LIN {X 0,Y 523.988,Z 418.315,A -85,B 0,C 180,E1 -4858.463,E2 -4858.463} C_VEL
LIN {X 0,Y 524.311,Z 419.919,A -85,B 0,C 180,E1 -4858.848,E2 -4858.848} C_VEL
LIN {X 0,Y 524.202,Z 424.484,A -85,B 0,C 180,E1 -4859.928,E2 -4859.928} C_VEL
LIN {X 0,Y 525.991,Z 433.873,A -85,B 0,C 180,E1 -4860.12,E2 -4860.12} C_VEL
LIN {X 0,Y 525.479,Z 529.837,A -85,B 0,C 180,E1 -4861.485,E2 -4861.485} C_VEL
LIN {X 0,Y 525.253,Z 542.81,A -85,B 0,C 180,E1 -4861.821,E2 -4861.821} C_VEL
LIN {X 0,Y 525.093,Z 555.331,A -85,B 0,C 180,E1 -4862.301,E2 -4862.301} C_VEL
LIN {X 0,Y 524.836,Z 568.104,A -85,B 0,C 180,E1 -4862.974,E2 -4862.974} C_VEL
LIN {X 0,Y 524.493,Z 579.334,A -85,B 0,C 180,E1 -4863.745,E2 -4863.745} C_VEL
LIN {X 0,Y 524.25,Z 589.443,A -85,B 0,C 180,E1 -4864.614,E2 -4864.614} C_VEL
LIN {X 0,Y 524.02,Z 598.626,A -85,B 0,C 180,E1 -4865.58,E2 -4865.58} C_VEL
LIN {X 0,Y 523.843,Z 606.368,A -85,B 0,C 180,E1 -4866.58,E2 -4866.58} C_VEL
LIN {X 0,Y 523.721,Z 613.507,A -85,B 0,C 180,E1 -4867.712,E2 -4867.712} C_VEL
LIN {X 0,Y 523.534,Z 619.416,A -85,B 0,C 180,E1 -4868.881,E2 -4868.881} C_VEL
LIN {X 0,Y 523.46,Z 624.093,A -85,B 0,C 180,E1 -4870.052,E2 -4870.052} C_VEL
LIN {X 0,Y 523.411,Z 628.198,A -85,B 0,C 180,E1 -4871.42,E2 -4871.42} C_VEL
LIN {X 0,Y 523.321,Z 630.26,A -85,B 0,C 180,E1 -4872.408,E2 -4872.408} C_VEL
LIN {X 0,Y 523.324,Z 632.229,A -85,B 0,C 180,E1 -4873.989,E2 -4873.989} C_VEL
LIN {X 0,Y 523.299,Z 632.553,A -85,B 0,C 180,E1 -4874.784,E2 -4874.784} C_VEL
LIN {X 0,Y 523.254,Z 631.982,A -85,B 0,C 180,E1 -4876.383,E2 -4876.383} C_VEL
LIN {X 0,Y 523.312,Z 630.501,A -85,B 0,C 180,E1 -4877.536,E2 -4877.536} C_VEL
LIN {X 0,Y 523.374,Z 626.71,A -85,B 0,C 180,E1 -4879.208,E2 -4879.208} C_VEL
LIN {X 0,Y 523.466,Z 622.639,A -85,B 0,C 180,E1 -4880.431,E2 -4880.431} C_VEL
LIN {X 0,Y 523.581,Z 616.177,A -85,B 0,C 180,E1 -4881.869,E2 -4881.869} C_VEL
LIN {X 0,Y 523.697,Z 610.264,A -85,B 0,C 180,E1 -4882.903,E2 -4882.903} C_VEL
LIN {X 0,Y 523.919,Z 602.842,A -85,B 0,C 180,E1 -4883.966,E2 -4883.966} C_VEL
LIN {X 0,Y 524.086,Z 596.098,A -85,B 0,C 180,E1 -4884.775,E2 -4884.775} C_VEL
LIN {X 0,Y 524.315,Z 587.958,A -85,B 0,C 180,E1 -4885.601,E2 -4885.601} C_VEL
LIN {X 0,Y 524.554,Z 577.757,A -85,B 0,C 180,E1 -4886.454,E2 -4886.454} C_VEL
LIN {X 0,Y 524.832,Z 566.75,A -85,B 0,C 180,E1 -4887.192,E2 -4887.192} C_VEL
LIN {X 0,Y 525.129,Z 555.209,A -85,B 0,C 180,E1 -4887.789,E2 -4887.789} C_VEL
LIN {X 0,Y 525.296,Z 542.798,A -85,B 0,C 180,E1 -4888.267,E2 -4888.267} C_VEL
LIN {X 0,Y 525.449,Z 530.555,A -85,B 0,C 180,E1 -4888.593,E2 -4888.593} C_VEL
LIN {X 0,Y 525.677,Z 483.88,A -85,B 0,C 180,E1 -4889.263,E2 -4889.263} C_VEL
LIN {X 0,Y 525.84,Z 432.621,A -85,B 0,C 180,E1 -4889.982,E2 -4889.982} C_VEL
LIN {X 0,Y 525.253,Z 429.53,A -85,B 0,C 180,E1 -4890.045,E2 -4890.045} C_VEL
LIN {X 0,Y 524.217,Z 426.571,A -85,B 0,C 180,E1 -4890.171,E2 -4890.171} C_VEL
LIN {X 0,Y 521.978,Z 423.441,A -85,B 0,C 180,E1 -4890.485,E2 -4890.485} C_VEL
LIN {X 0,Y 519.924,Z 421.666,A -85,B 0,C 180,E1 -4890.834,E2 -4890.834} C_VEL
LIN {X 0,Y 517.617,Z 419.8,A -85,B 0,C 180,E1 -4891.394,E2 -4891.394} C_VEL
LIN {X 0,Y 516.936,Z 419.124,A -85,B 0,C 180,E1 -4891.783,E2 -4891.783} C_VEL
LIN {X 0,Y 516.908,Z 419.099,A -85,B 0,C 180,E1 -4891.864,E2 -4891.864} C_VEL
LIN {X 0,Y 516.875,Z 419.099,A -85,B 0,C 180,E1 -4894.825,E2 -4894.825} C_VEL
LIN {X 0,Y 516.867,Z 419.099,A -85,B 0,C 180,E1 -4897.94,E2 -4897.94} C_VEL
LIN {X 0,Y 516.856,Z 419.102,A -85,B 0,C 180,E1 -4900.744,E2 -4900.744} C_VEL
LIN {X 0,Y 516.884,Z 419.097,A -85,B 0,C 180,E1 -4903.903,E2 -4903.903} C_VEL
LIN {X 0,Y 516.882,Z 419.099,A -85,B 0,C 180,E1 -4906.107,E2 -4906.107} C_VEL
LIN {X 0,Y 516.854,Z 419.098,A -85,B 0,C 180,E1 -4909.255,E2 -4909.255} C_VEL
LIN {X 0,Y 516.864,Z 419.101,A -85,B 0,C 180,E1 -4912.06,E2 -4912.06} C_VEL
LIN {X 0,Y 516.876,Z 419.096,A -85,B 0,C 180,E1 -4915.174,E2 -4915.174} C_VEL
LIN {X 0,Y 516.875,Z 419.098,A -85,B 0,C 180,E1 -4917.975,E2 -4917.975} C_VEL
LIN {X 0,Y 516.906,Z 419.097,A -85,B 0,C 180,E1 -4920.694,E2 -4920.694} C_VEL
LIN {X 0,Y 516.89,Z 419.095,A -85,B 0,C 180,E1 -4923.816,E2 -4923.816} C_VEL
LIN {X 0,Y 516.86,Z 419.102,A -85,B 0,C 180,E1 -4926.776,E2 -4926.776} C_VEL
LIN {X 0,Y 516.94,Z 419.088,A -85,B 0,C 180,E1 -4929.732,E2 -4929.732} C_VEL
LIN {X 0,Y 516.887,Z 419.101,A -85,B 0,C 180,E1 -4932.594,E2 -4932.594} C_VEL
LIN {X 0,Y 516.938,Z 419.089,A -85,B 0,C 180,E1 -4935.03,E2 -4935.03} C_VEL
LIN {X 0,Y 516.969,Z 419.089,A -85,B 0,C 180,E1 -4938.233,E2 -4938.233} C_VEL
LIN {X 0,Y 516.955,Z 419.085,A -85,B 0,C 180,E1 -4941.399,E2 -4941.399} C_VEL
LIN {X 0,Y 517.014,Z 419.087,A -85,B 0,C 180,E1 -4944.54,E2 -4944.54} C_VEL
LIN {X 0,Y 517.082,Z 419.07,A -85,B 0,C 180,E1 -4947.663,E2 -4947.663} C_VEL
LIN {X 0,Y 517.092,Z 419.073,A -85,B 0,C 180,E1 -4950.778,E2 -4950.778} C_VEL
LIN {X 0,Y 516.974,Z 419.084,A -85,B 0,C 180,E1 -4953.117,E2 -4953.117} C_VEL
LIN {X 0,Y 517.008,Z 419.084,A -85,B 0,C 180,E1 -4956.243,E2 -4956.243} C_VEL
LIN {X 0,Y 516.94,Z 419.087,A -85,B 0,C 180,E1 -4959.389,E2 -4959.389} C_VEL
LIN {X 0,Y 516.954,Z 419.086,A -85,B 0,C 180,E1 -4961.807,E2 -4961.807} C_VEL
LIN {X 0,Y 516.949,Z 419.087,A -85,B 0,C 180,E1 -4965.147,E2 -4965.147} C_VEL
LIN {X 0,Y 516.917,Z 419.095,A -85,B 0,C 180,E1 -4968.222,E2 -4968.222} C_VEL
LIN {X 0,Y 516.913,Z 419.097,A -85,B 0,C 180,E1 -4970.701,E2 -4970.701} C_VEL
LIN {X 0,Y 516.891,Z 419.096,A -85,B 0,C 180,E1 -4974.073,E2 -4974.073} C_VEL
LIN {X 0,Y 516.897,Z 419.1,A -85,B 0,C 180,E1 -4976.659,E2 -4976.659} C_VEL
LIN {X 0,Y 516.91,Z 419.091,A -85,B 0,C 180,E1 -4979.523,E2 -4979.523} C_VEL
LIN {X 0,Y 516.896,Z 419.102,A -85,B 0,C 180,E1 -4982.543,E2 -4982.543} C_VEL
LIN {X 0,Y 516.864,Z 419.097,A -85,B 0,C 180,E1 -4985.329,E2 -4985.329} C_VEL
LIN {X 0,Y 516.878,Z 419.096,A -85,B 0,C 180,E1 -4987.943,E2 -4987.943} C_VEL
LIN {X 0,Y 516.881,Z 419.101,A -85,B 0,C 180,E1 -4990.742,E2 -4990.742} C_VEL
LIN {X 0,Y 516.88,Z 419.096,A -85,B 0,C 180,E1 -4993.903,E2 -4993.903} C_VEL
LIN {X 0,Y 516.88,Z 419.097,A -85,B 0,C 180,E1 -4996.107,E2 -4996.107} C_VEL
LIN {X 0,Y 516.881,Z 419.095,A -85,B 0,C 180,E1 -4999.258,E2 -4999.258} C_VEL
LIN {X 0,Y 516.86,Z 419.102,A -85,B 0,C 180,E1 -5002.274,E2 -5002.274} C_VEL
LIN {X 0,Y 516.881,Z 419.096,A -85,B 0,C 180,E1 -5005.175,E2 -5005.175} C_VEL
LIN {X 0,Y 516.873,Z 419.097,A -85,B 0,C 180,E1 -5007.975,E2 -5007.975} C_VEL
LIN {X 0,Y 516.92,Z 419.098,A -85,B 0,C 180,E1 -5010.695,E2 -5010.695} C_VEL
LIN {X 0,Y 516.911,Z 419.091,A -85,B 0,C 180,E1 -5013.811,E2 -5013.811} C_VEL
LIN {X 0,Y 516.86,Z 419.104,A -85,B 0,C 180,E1 -5016.776,E2 -5016.776} C_VEL
LIN {X 0,Y 516.939,Z 419.087,A -85,B 0,C 180,E1 -5019.732,E2 -5019.732} C_VEL
LIN {X 0,Y 516.905,Z 419.101,A -85,B 0,C 180,E1 -5022.595,E2 -5022.595} C_VEL
LIN {X 0,Y 516.941,Z 419.09,A -85,B 0,C 180,E1 -5025.03,E2 -5025.03} C_VEL
LIN {X 0,Y 516.966,Z 419.087,A -85,B 0,C 180,E1 -5028.234,E2 -5028.234} C_VEL
LIN {X 0,Y 516.965,Z 419.085,A -85,B 0,C 180,E1 -5031.4,E2 -5031.4} C_VEL
LIN {X 0,Y 517.025,Z 419.085,A -85,B 0,C 180,E1 -5034.54,E2 -5034.54} C_VEL
LIN {X 0,Y 517.083,Z 419.069,A -85,B 0,C 180,E1 -5037.663,E2 -5037.663} C_VEL
LIN {X 0,Y 517.093,Z 419.076,A -85,B 0,C 180,E1 -5040.779,E2 -5040.779} C_VEL
LIN {X 0,Y 517.009,Z 419.081,A -85,B 0,C 180,E1 -5043.117,E2 -5043.117} C_VEL
LIN {X 0,Y 517.008,Z 419.082,A -85,B 0,C 180,E1 -5046.243,E2 -5046.243} C_VEL
LIN {X 0,Y 516.944,Z 419.087,A -85,B 0,C 180,E1 -5049.389,E2 -5049.389} C_VEL
LIN {X 0,Y 516.952,Z 419.086,A -85,B 0,C 180,E1 -5051.807,E2 -5051.807} C_VEL
LIN {X 0,Y 516.948,Z 419.089,A -85,B 0,C 180,E1 -5055.148,E2 -5055.148} C_VEL
LIN {X 0,Y 516.916,Z 419.093,A -85,B 0,C 180,E1 -5058.223,E2 -5058.223} C_VEL
LIN {X 0,Y 516.912,Z 419.1,A -85,B 0,C 180,E1 -5060.702,E2 -5060.702} C_VEL
LIN {X 0,Y 516.902,Z 419.093,A -85,B 0,C 180,E1 -5064.073,E2 -5064.073} C_VEL
LIN {X 0,Y 516.904,Z 419.101,A -85,B 0,C 180,E1 -5066.659,E2 -5066.659} C_VEL
LIN {X 0,Y 516.911,Z 419.091,A -85,B 0,C 180,E1 -5069.524,E2 -5069.524} C_VEL
LIN {X 0,Y 516.895,Z 419.099,A -85,B 0,C 180,E1 -5072.543,E2 -5072.543} C_VEL
LIN {X 0,Y 516.867,Z 419.098,A -85,B 0,C 180,E1 -5075.33,E2 -5075.33} C_VEL
LIN {X 0,Y 516.88,Z 419.095,A -85,B 0,C 180,E1 -5077.943,E2 -5077.943} C_VEL
LIN {X 0,Y 516.883,Z 419.104,A -85,B 0,C 180,E1 -5080.742,E2 -5080.742} C_VEL
LIN {X 0,Y 516.883,Z 419.102,A -85,B 0,C 180,E1 -5082.832,E2 -5082.832} C_VEL
LIN {X 0,Y 516.924,Z 419.094,A -85,B 0,C 180,E1 -5085.01,E2 -5085.01} C_VEL
LIN {X 0,Y 516.914,Z 419.095,A -85,B 0,C 180,E1 -5088.399,E2 -5088.399} C_VEL
LIN {X 0,Y 516.882,Z 419.096,A -85,B 0,C 180,E1 -5091.284,E2 -5091.284} C_VEL
LIN {X 0,Y 516.869,Z 419.098,A -85,B 0,C 180,E1 -5094.22,E2 -5094.22} C_VEL
LIN {X 0,Y 516.896,Z 419.098,A -85,B 0,C 180,E1 -5097.053,E2 -5097.053} C_VEL
LIN {X 0,Y 516.893,Z 419.094,A -85,B 0,C 180,E1 -5099.797,E2 -5099.797} C_VEL
LIN {X 0,Y 516.925,Z 419.097,A -85,B 0,C 180,E1 -5102.467,E2 -5102.467} C_VEL
LIN {X 0,Y 516.954,Z 419.122,A -85,B 0,C 180,E1 -5103.438,E2 -5103.438} C_VEL
LIN {X 0,Y 519.032,Z 430.297,A -85,B 0,C 180,E1 -5105.181,E2 -5105.181} C_VEL
LIN {X 0,Y 518.58,Z 445.899,A -85,B 0,C 180,E1 -5107.421,E2 -5107.421} C_VEL
LIN {X 0,Y 518.088,Z 466.974,A -85,B 0,C 180,E1 -5110.383,E2 -5110.383} C_VEL
LIN {X 0,Y 517.598,Z 488.869,A -85,B 0,C 180,E1 -5113.433,E2 -5113.433} C_VEL
LIN {X 0,Y 517.403,Z 497.471,A -85,B 0,C 180,E1 -5114.627,E2 -5114.627} C_VEL
LIN {X 0,Y 518.961,Z 510.132,A -85,B 0,C 180,E1 -5114.873,E2 -5114.873} C_VEL
LIN {X 0,Y 518.553,Z 604.493,A -85,B 0,C 180,E1 -5116.205,E2 -5116.205} C_VEL
LIN {X 0,Y 518.352,Z 617.14,A -85,B 0,C 180,E1 -5116.5,E2 -5116.5} C_VEL
LIN {X 0,Y 518.062,Z 630.067,A -85,B 0,C 180,E1 -5116.966,E2 -5116.966} C_VEL
LIN {X 0,Y 517.822,Z 642.684,A -85,B 0,C 180,E1 -5117.594,E2 -5117.594} C_VEL
LIN {X 0,Y 517.526,Z 654.284,A -85,B 0,C 180,E1 -5118.346,E2 -5118.346} C_VEL
LIN {X 0,Y 517.212,Z 665.109,A -85,B 0,C 180,E1 -5119.232,E2 -5119.232} C_VEL
LIN {X 0,Y 516.948,Z 674.862,A -85,B 0,C 180,E1 -5120.216,E2 -5120.216} C_VEL
LIN {X 0,Y 516.739,Z 682.861,A -85,B 0,C 180,E1 -5121.199,E2 -5121.199} C_VEL
LIN {X 0,Y 516.555,Z 690.676,A -85,B 0,C 180,E1 -5122.377,E2 -5122.377} C_VEL
LIN {X 0,Y 516.421,Z 696.438,A -85,B 0,C 180,E1 -5123.446,E2 -5123.446} C_VEL
LIN {X 0,Y 516.402,Z 701.206,A -85,B 0,C 180,E1 -5124.534,E2 -5124.534} C_VEL
LIN {X 0,Y 516.331,Z 705.226,A -85,B 0,C 180,E1 -5125.707,E2 -5125.707} C_VEL
LIN {X 0,Y 516.282,Z 708.192,A -85,B 0,C 180,E1 -5126.879,E2 -5126.879} C_VEL
LIN {X 0,Y 516.261,Z 709.605,A -85,B 0,C 180,E1 -5127.66,E2 -5127.66} C_VEL
LIN {X 0,Y 516.169,Z 711.22,A -85,B 0,C 180,E1 -5129.22,E2 -5129.22} C_VEL
LIN {X 0,Y 516.167,Z 711.435,A -85,B 0,C 180,E1 -5130,E2 -5130} C_VEL
LIN {X 0,Y 516.17,Z 711.214,A -85,B 0,C 180,E1 -5130.78,E2 -5130.78} C_VEL
LIN {X 0,Y 516.261,Z 709.591,A -85,B 0,C 180,E1 -5132.341,E2 -5132.341} C_VEL
LIN {X 0,Y 516.296,Z 708.169,A -85,B 0,C 180,E1 -5133.122,E2 -5133.122} C_VEL
LIN {X 0,Y 516.348,Z 705.187,A -85,B 0,C 180,E1 -5134.293,E2 -5134.293} C_VEL
LIN {X 0,Y 516.402,Z 701.146,A -85,B 0,C 180,E1 -5135.467,E2 -5135.467} C_VEL
LIN {X 0,Y 516.484,Z 695.108,A -85,B 0,C 180,E1 -5136.803,E2 -5136.803} C_VEL
LIN {X 0,Y 516.606,Z 688.128,A -85,B 0,C 180,E1 -5138.016,E2 -5138.016} C_VEL
LIN {X 0,Y 516.8,Z 679.686,A -85,B 0,C 180,E1 -5139.195,E2 -5139.195} C_VEL
LIN {X 0,Y 517.041,Z 671.016,A -85,B 0,C 180,E1 -5140.178,E2 -5140.178} C_VEL
LIN {X 0,Y 517.331,Z 660.315,A -85,B 0,C 180,E1 -5141.163,E2 -5141.163} C_VEL
LIN {X 0,Y 517.576,Z 649.28,A -85,B 0,C 180,E1 -5141.98,E2 -5141.98} C_VEL
LIN {X 0,Y 517.929,Z 637.022,A -85,B 0,C 180,E1 -5142.689,E2 -5142.689} C_VEL
LIN {X 0,Y 518.168,Z 624.585,A -85,B 0,C 180,E1 -5143.231,E2 -5143.231} C_VEL
LIN {X 0,Y 518.419,Z 611.883,A -85,B 0,C 180,E1 -5143.624,E2 -5143.624} C_VEL
LIN {X 0,Y 518.649,Z 597.089,A -85,B 0,C 180,E1 -5143.893,E2 -5143.893} C_VEL
LIN {X 0,Y 518.808,Z 507.894,A -85,B 0,C 180,E1 -5145.156,E2 -5145.156} C_VEL
LIN {X 0,Y 517.345,Z 496.789,A -85,B 0,C 180,E1 -5145.376,E2 -5145.376} C_VEL
LIN {X 0,Y 517.74,Z 476.234,A -85,B 0,C 180,E1 -5148.193,E2 -5148.193} C_VEL
LIN {X 0,Y 518.264,Z 454.035,A -85,B 0,C 180,E1 -5151.269,E2 -5151.269} C_VEL
LIN {X 0,Y 518.756,Z 431.819,A -85,B 0,C 180,E1 -5154.407,E2 -5154.407} C_VEL
LIN {X 0,Y 518.806,Z 428.851,A -85,B 0,C 180,E1 -5154.831,E2 -5154.831} C_VEL
LIN {X 0,Y 516.94,Z 419.094,A -85,B 0,C 180,E1 -5156.352,E2 -5156.352} C_VEL
LIN {X 0,Y 516.915,Z 419.098,A -85,B 0,C 180,E1 -5159.524,E2 -5159.524} C_VEL
LIN {X 0,Y 516.9,Z 419.1,A -85,B 0,C 180,E1 -5162.544,E2 -5162.544} C_VEL
LIN {X 0,Y 516.872,Z 419.103,A -85,B 0,C 180,E1 -5165.33,E2 -5165.33} C_VEL
LIN {X 0,Y 516.884,Z 419.096,A -85,B 0,C 180,E1 -5167.943,E2 -5167.943} C_VEL
LIN {X 0,Y 516.887,Z 419.102,A -85,B 0,C 180,E1 -5170.742,E2 -5170.742} C_VEL
LIN {X 0,Y 516.886,Z 419.104,A -85,B 0,C 180,E1 -5172.832,E2 -5172.832} C_VEL
LIN {X 0,Y 516.899,Z 419.098,A -85,B 0,C 180,E1 -5175.007,E2 -5175.007} C_VEL
LIN {X 0,Y 516.914,Z 419.097,A -85,B 0,C 180,E1 -5178.399,E2 -5178.399} C_VEL
LIN {X 0,Y 516.883,Z 419.096,A -85,B 0,C 180,E1 -5181.284,E2 -5181.284} C_VEL
LIN {X 0,Y 516.87,Z 419.101,A -85,B 0,C 180,E1 -5184.219,E2 -5184.219} C_VEL
LIN {X 0,Y 516.899,Z 419.094,A -85,B 0,C 180,E1 -5187.053,E2 -5187.053} C_VEL
LIN {X 0,Y 516.871,Z 419.098,A -85,B 0,C 180,E1 -5189.795,E2 -5189.795} C_VEL
LIN {X 0,Y 516.877,Z 419.104,A -85,B 0,C 180,E1 -5192.464,E2 -5192.464} C_VEL
LIN {X 0,Y 516.848,Z 419.101,A -85,B 0,C 180,E1 -5195.069,E2 -5195.069} C_VEL
LIN {X 0,Y 516.873,Z 419.099,A -85,B 0,C 180,E1 -5197.622,E2 -5197.622} C_VEL
LIN {X 0,Y 516.866,Z 419.105,A -85,B 0,C 180,E1 -5200.127,E2 -5200.127} C_VEL
LIN {X 0,Y 516.867,Z 419.1,A -85,B 0,C 180,E1 -5202.594,E2 -5202.594} C_VEL
LIN {X 0,Y 516.857,Z 419.106,A -85,B 0,C 180,E1 -5205.832,E2 -5205.832} C_VEL
LIN {X 0,Y 516.923,Z 419.097,A -85,B 0,C 180,E1 -5208.233,E2 -5208.233} C_VEL
LIN {X 0,Y 516.92,Z 419.095,A -85,B 0,C 180,E1 -5211.399,E2 -5211.399} C_VEL
LIN {X 0,Y 516.98,Z 419.087,A -85,B 0,C 180,E1 -5214.539,E2 -5214.539} C_VEL
LIN {X 0,Y 517.025,Z 419.086,A -85,B 0,C 180,E1 -5218.052,E2 -5218.052} C_VEL
LIN {X 0,Y 517.007,Z 419.337,A -85,B 0,C 180,E1 -5218.345,E2 -5218.345} C_VEL
LIN {X 0,Y 517.28,Z 423.009,A -85,B 0,C 180,E1 -5219.221,E2 -5219.221} C_VEL
LIN {X 0,Y 517.308,Z 425.389,A -85,B 0,C 180,E1 -5219.732,E2 -5219.732} C_VEL
LIN {X 0,Y 519.149,Z 434.62,A -85,B 0,C 180,E1 -5219.927,E2 -5219.927} C_VEL
LIN {X 0,Y 518.51,Z 531.284,A -85,B 0,C 180,E1 -5221.335,E2 -5221.335} C_VEL
LIN {X 0,Y 518.342,Z 544.694,A -85,B 0,C 180,E1 -5221.7,E2 -5221.7} C_VEL
LIN {X 0,Y 518.14,Z 556.874,A -85,B 0,C 180,E1 -5222.186,E2 -5222.186} C_VEL
LIN {X 0,Y 517.904,Z 568.571,A -85,B 0,C 180,E1 -5222.82,E2 -5222.82} C_VEL
LIN {X 0,Y 517.551,Z 579.85,A -85,B 0,C 180,E1 -5223.601,E2 -5223.601} C_VEL
LIN {X 0,Y 517.273,Z 589.985,A -85,B 0,C 180,E1 -5224.481,E2 -5224.481} C_VEL
LIN {X 0,Y 517.038,Z 599.151,A -85,B 0,C 180,E1 -5225.46,E2 -5225.46} C_VEL
LIN {X 0,Y 516.797,Z 607.986,A -85,B 0,C 180,E1 -5226.632,E2 -5226.632} C_VEL
LIN {X 0,Y 516.641,Z 615.138,A -85,B 0,C 180,E1 -5227.818,E2 -5227.818} C_VEL
LIN {X 0,Y 516.488,Z 620.854,A -85,B 0,C 180,E1 -5229.003,E2 -5229.003} C_VEL
LIN {X 0,Y 516.4,Z 625.362,A -85,B 0,C 180,E1 -5230.191,E2 -5230.191} C_VEL
LIN {X 0,Y 516.302,Z 629.7,A -85,B 0,C 180,E1 -5231.782,E2 -5231.782} C_VEL
LIN {X 0,Y 516.24,Z 631.194,A -85,B 0,C 180,E1 -5232.581,E2 -5232.581} C_VEL
LIN {X 0,Y 516.244,Z 632.889,A -85,B 0,C 180,E1 -5234.185,E2 -5234.185} C_VEL
LIN {X 0,Y 516.21,Z 633.139,A -85,B 0,C 180,E1 -5234.992,E2 -5234.992} C_VEL
LIN {X 0,Y 516.195,Z 632.919,A -85,B 0,C 180,E1 -5235.801,E2 -5235.801} C_VEL
LIN {X 0,Y 516.241,Z 631.278,A -85,B 0,C 180,E1 -5237.428,E2 -5237.428} C_VEL
LIN {X 0,Y 516.296,Z 628.843,A -85,B 0,C 180,E1 -5238.656,E2 -5238.656} C_VEL
LIN {X 0,Y 516.357,Z 625.294,A -85,B 0,C 180,E1 -5239.893,E2 -5239.893} C_VEL
LIN {X 0,Y 516.445,Z 620.518,A -85,B 0,C 180,E1 -5241.138,E2 -5241.138} C_VEL
LIN {X 0,Y 516.605,Z 614.367,A -85,B 0,C 180,E1 -5242.391,E2 -5242.391} C_VEL
LIN {X 0,Y 516.818,Z 606.511,A -85,B 0,C 180,E1 -5243.651,E2 -5243.651} C_VEL
LIN {X 0,Y 517.042,Z 597.84,A -85,B 0,C 180,E1 -5244.76,E2 -5244.76} C_VEL
LIN {X 0,Y 517.309,Z 589.228,A -85,B 0,C 180,E1 -5245.661,E2 -5245.661} C_VEL
LIN {X 0,Y 517.54,Z 579.353,A -85,B 0,C 180,E1 -5246.513,E2 -5246.513} C_VEL
LIN {X 0,Y 517.846,Z 568.558,A -85,B 0,C 180,E1 -5247.261,E2 -5247.261} C_VEL
LIN {X 0,Y 518.187,Z 556.468,A -85,B 0,C 180,E1 -5247.915,E2 -5247.915} C_VEL
LIN {X 0,Y 518.404,Z 544.005,A -85,B 0,C 180,E1 -5248.409,E2 -5248.409} C_VEL
LIN {X 0,Y 518.543,Z 531.159,A -85,B 0,C 180,E1 -5248.76,E2 -5248.76} C_VEL
LIN {X 0,Y 518.771,Z 491.313,A -85,B 0,C 180,E1 -5249.348,E2 -5249.348} C_VEL
LIN {X 0,Y 518.956,Z 433.244,A -85,B 0,C 180,E1 -5250.182,E2 -5250.182} C_VEL
LIN {X 0,Y 517.154,Z 424.213,A -85,B 0,C 180,E1 -5250.384,E2 -5250.384} C_VEL
LIN {X 0,Y 516.963,Z 419.316,A -85,B 0,C 180,E1 -5251.497,E2 -5251.497} C_VEL
LIN {X 0,Y 516.908,Z 419.099,A -85,B 0,C 180,E1 -5251.864,E2 -5251.864} C_VEL
LIN {X 0,Y 516.206,Z 419.188,A -85,B 0,C 180,E1 -5252.514,E2 -5252.514} C_VEL
LIN {X 0,Y 513.315,Z 419.546,A -85,B 0,C 180,E1 -5253.57,E2 -5253.57} C_VEL
LIN {X 0,Y 510.903,Z 419.848,A -85,B 0,C 180,E1 -5254.42,E2 -5254.42} C_VEL
LIN {X 0,Y 509.889,Z 419.968,A -85,B 0,C 180,E1 -5255.077,E2 -5255.077} C_VEL
LIN {X 0,Y 509.816,Z 419.976,A -85,B 0,C 180,E1 -5255.299,E2 -5255.299} C_VEL
LIN {X 0,Y 509.819,Z 419.983,A -85,B 0,C 180,E1 -5258.341,E2 -5258.341} C_VEL
LIN {X 0,Y 509.834,Z 419.972,A -85,B 0,C 180,E1 -5261.428,E2 -5261.428} C_VEL
LIN {X 0,Y 509.842,Z 419.977,A -85,B 0,C 180,E1 -5264.67,E2 -5264.67} C_VEL
LIN {X 0,Y 509.793,Z 419.978,A -85,B 0,C 180,E1 -5267.505,E2 -5267.505} C_VEL
LIN {X 0,Y 509.834,Z 419.978,A -85,B 0,C 180,E1 -5270.646,E2 -5270.646} C_VEL
LIN {X 0,Y 509.783,Z 419.979,A -85,B 0,C 180,E1 -5273.643,E2 -5273.643} C_VEL
LIN {X 0,Y 509.854,Z 419.978,A -85,B 0,C 180,E1 -5276.538,E2 -5276.538} C_VEL
LIN {X 0,Y 509.836,Z 419.972,A -85,B 0,C 180,E1 -5279.333,E2 -5279.333} C_VEL
LIN {X 0,Y 509.838,Z 419.976,A -85,B 0,C 180,E1 -5282.051,E2 -5282.051} C_VEL
LIN {X 0,Y 509.808,Z 419.981,A -85,B 0,C 180,E1 -5284.7,E2 -5284.7} C_VEL
LIN {X 0,Y 509.828,Z 419.973,A -85,B 0,C 180,E1 -5287.458,E2 -5287.458} C_VEL
LIN {X 0,Y 509.917,Z 419.964,A -85,B 0,C 180,E1 -5289.844,E2 -5289.844} C_VEL
LIN {X 0,Y 509.849,Z 419.971,A -85,B 0,C 180,E1 -5293.173,E2 -5293.173} C_VEL
LIN {X 0,Y 509.854,Z 419.97,A -85,B 0,C 180,E1 -5295.634,E2 -5295.634} C_VEL
LIN {X 0,Y 509.914,Z 419.966,A -85,B 0,C 180,E1 -5298.874,E2 -5298.874} C_VEL
LIN {X 0,Y 509.91,Z 419.966,A -85,B 0,C 180,E1 -5302.077,E2 -5302.077} C_VEL
LIN {X 0,Y 509.965,Z 419.966,A -85,B 0,C 180,E1 -5304.464,E2 -5304.464} C_VEL
LIN {X 0,Y 510.051,Z 419.945,A -85,B 0,C 180,E1 -5307.631,E2 -5307.631} C_VEL
LIN {X 0,Y 510.062,Z 419.949,A -85,B 0,C 180,E1 -5310.789,E2 -5310.789} C_VEL
LIN {X 0,Y 509.918,Z 419.963,A -85,B 0,C 180,E1 -5313.16,E2 -5313.16} C_VEL
LIN {X 0,Y 509.977,Z 419.961,A -85,B 0,C 180,E1 -5316.329,E2 -5316.329} C_VEL
LIN {X 0,Y 509.88,Z 419.967,A -85,B 0,C 180,E1 -5319.52,E2 -5319.52} C_VEL
LIN {X 0,Y 509.906,Z 419.965,A -85,B 0,C 180,E1 -5321.931,E2 -5321.931} C_VEL
LIN {X 0,Y 509.896,Z 419.965,A -85,B 0,C 180,E1 -5325.241,E2 -5325.241} C_VEL
LIN {X 0,Y 509.862,Z 419.978,A -85,B 0,C 180,E1 -5328.483,E2 -5328.483} C_VEL
LIN {X 0,Y 509.851,Z 419.973,A -85,B 0,C 180,E1 -5331.001,E2 -5331.001} C_VEL
LIN {X 0,Y 509.823,Z 419.974,A -85,B 0,C 180,E1 -5333.564,E2 -5333.564} C_VEL
LIN {X 0,Y 509.879,Z 419.974,A -85,B 0,C 180,E1 -5336.371,E2 -5336.371} C_VEL
LIN {X 0,Y 509.859,Z 419.97,A -85,B 0,C 180,E1 -5339.726,E2 -5339.726} C_VEL
LIN {X 0,Y 509.873,Z 419.973,A -85,B 0,C 180,E1 -5342.774,E2 -5342.774} C_VEL
LIN {X 0,Y 509.823,Z 419.974,A -85,B 0,C 180,E1 -5345.578,E2 -5345.578} C_VEL
LIN {X 0,Y 509.848,Z 419.977,A -85,B 0,C 180,E1 -5348.338,E2 -5348.338} C_VEL
LIN {X 0,Y 509.852,Z 419.97,A -85,B 0,C 180,E1 -5351.426,E2 -5351.426} C_VEL
LIN {X 0,Y 509.838,Z 419.98,A -85,B 0,C 180,E1 -5354.67,E2 -5354.67} C_VEL
LIN {X 0,Y 509.849,Z 419.973,A -85,B 0,C 180,E1 -5358.104,E2 -5358.104} C_VEL
LIN {X 0,Y 509.845,Z 419.979,A -85,B 0,C 180,E1 -5360.647,E2 -5360.647} C_VEL
LIN {X 0,Y 509.808,Z 419.976,A -85,B 0,C 180,E1 -5363.645,E2 -5363.645} C_VEL
LIN {X 0,Y 509.858,Z 419.978,A -85,B 0,C 180,E1 -5366.539,E2 -5366.539} C_VEL
LIN {X 0,Y 509.845,Z 419.972,A -85,B 0,C 180,E1 -5369.334,E2 -5369.334} C_VEL
LIN {X 0,Y 509.882,Z 419.968,A -85,B 0,C 180,E1 -5372.054,E2 -5372.054} C_VEL
LIN {X 0,Y 509.824,Z 419.982,A -85,B 0,C 180,E1 -5374.701,E2 -5374.701} C_VEL
LIN {X 0,Y 509.826,Z 419.974,A -85,B 0,C 180,E1 -5377.458,E2 -5377.458} C_VEL
LIN {X 0,Y 509.916,Z 419.963,A -85,B 0,C 180,E1 -5379.845,E2 -5379.845} C_VEL
LIN {X 0,Y 509.87,Z 419.97,A -85,B 0,C 180,E1 -5383.174,E2 -5383.174} C_VEL
LIN {X 0,Y 509.861,Z 419.969,A -85,B 0,C 180,E1 -5385.634,E2 -5385.634} C_VEL
LIN {X 0,Y 509.912,Z 419.968,A -85,B 0,C 180,E1 -5388.875,E2 -5388.875} C_VEL
LIN {X 0,Y 509.951,Z 419.96,A -85,B 0,C 180,E1 -5392.078,E2 -5392.078} C_VEL
LIN {X 0,Y 509.976,Z 419.961,A -85,B 0,C 180,E1 -5394.464,E2 -5394.464} C_VEL
LIN {X 0,Y 510.054,Z 419.945,A -85,B 0,C 180,E1 -5397.631,E2 -5397.631} C_VEL
LIN {X 0,Y 510.063,Z 419.951,A -85,B 0,C 180,E1 -5400.79,E2 -5400.79} C_VEL
LIN {X 0,Y 509.95,Z 419.96,A -85,B 0,C 180,E1 -5403.16,E2 -5403.16} C_VEL
LIN {X 0,Y 509.977,Z 419.959,A -85,B 0,C 180,E1 -5406.33,E2 -5406.33} C_VEL
LIN {X 0,Y 509.911,Z 419.972,A -85,B 0,C 180,E1 -5408.72,E2 -5408.72} C_VEL
LIN {X 0,Y 509.905,Z 419.964,A -85,B 0,C 180,E1 -5411.932,E2 -5411.932} C_VEL
LIN {X 0,Y 509.894,Z 419.967,A -85,B 0,C 180,E1 -5415.242,E2 -5415.242} C_VEL
LIN {X 0,Y 509.867,Z 419.969,A -85,B 0,C 180,E1 -5417.993,E2 -5417.993} C_VEL
LIN {X 0,Y 509.887,Z 419.971,A -85,B 0,C 180,E1 -5420.402,E2 -5420.402} C_VEL
LIN {X 0,Y 509.829,Z 419.973,A -85,B 0,C 180,E1 -5423.564,E2 -5423.564} C_VEL
LIN {X 0,Y 509.886,Z 419.97,A -85,B 0,C 180,E1 -5426.373,E2 -5426.373} C_VEL
LIN {X 0,Y 509.872,Z 419.975,A -85,B 0,C 180,E1 -5428.845,E2 -5428.845} C_VEL
LIN {X 0,Y 509.82,Z 419.974,A -85,B 0,C 180,E1 -5431.59,E2 -5431.59} C_VEL
LIN {X 0,Y 509.848,Z 419.975,A -85,B 0,C 180,E1 -5434.414,E2 -5434.414} C_VEL
LIN {X 0,Y 509.817,Z 419.976,A -85,B 0,C 180,E1 -5437.341,E2 -5437.341} C_VEL
LIN {X 0,Y 509.838,Z 419.976,A -85,B 0,C 180,E1 -5440.382,E2 -5440.382} C_VEL
LIN {X 0,Y 509.823,Z 419.978,A -85,B 0,C 180,E1 -5443.062,E2 -5443.062} C_VEL
LIN {X 0,Y 509.831,Z 419.973,A -85,B 0,C 180,E1 -5445.793,E2 -5445.793} C_VEL
LIN {X 0,Y 509.856,Z 419.976,A -85,B 0,C 180,E1 -5448.575,E2 -5448.575} C_VEL
LIN {X 0,Y 509.851,Z 419.97,A -85,B 0,C 180,E1 -5451.787,E2 -5451.787} C_VEL
LIN {X 0,Y 509.828,Z 419.98,A -85,B 0,C 180,E1 -5454.622,E2 -5454.622} C_VEL
LIN {X 0,Y 509.862,Z 419.97,A -85,B 0,C 180,E1 -5457.481,E2 -5457.481} C_VEL
LIN {X 0,Y 509.86,Z 419.973,A -85,B 0,C 180,E1 -5460.274,E2 -5460.274} C_VEL
LIN {X 0,Y 509.939,Z 420.148,A -85,B 0,C 180,E1 -5463.258,E2 -5463.258} C_VEL
LIN {X 0,Y 512.148,Z 431.593,A -85,B 0,C 180,E1 -5465.071,E2 -5465.071} C_VEL
LIN {X 0,Y 511.609,Z 447.435,A -85,B 0,C 180,E1 -5467.379,E2 -5467.379} C_VEL
LIN {X 0,Y 511.109,Z 468.029,A -85,B 0,C 180,E1 -5470.313,E2 -5470.313} C_VEL
LIN {X 0,Y 510.548,Z 489.844,A -85,B 0,C 180,E1 -5473.403,E2 -5473.403} C_VEL
LIN {X 0,Y 510.369,Z 496.977,A -85,B 0,C 180,E1 -5474.407,E2 -5474.407} C_VEL
LIN {X 0,Y 512.09,Z 510.248,A -85,B 0,C 180,E1 -5474.674,E2 -5474.674} C_VEL
LIN {X 0,Y 511.66,Z 603.258,A -85,B 0,C 180,E1 -5476.016,E2 -5476.016} C_VEL
LIN {X 0,Y 511.438,Z 616.185,A -85,B 0,C 180,E1 -5476.313,E2 -5476.313} C_VEL
LIN {X 0,Y 511.134,Z 629.267,A -85,B 0,C 180,E1 -5476.786,E2 -5476.786} C_VEL
LIN {X 0,Y 510.88,Z 640.913,A -85,B 0,C 180,E1 -5477.364,E2 -5477.364} C_VEL
LIN {X 0,Y 510.565,Z 652.22,A -85,B 0,C 180,E1 -5478.084,E2 -5478.084} C_VEL
LIN {X 0,Y 510.229,Z 663.38,A -85,B 0,C 180,E1 -5478.982,E2 -5478.982} C_VEL
LIN {X 0,Y 509.904,Z 674.24,A -85,B 0,C 180,E1 -5480.079,E2 -5480.079} C_VEL
LIN {X 0,Y 509.68,Z 682.26,A -85,B 0,C 180,E1 -5481.076,E2 -5481.076} C_VEL
LIN {X 0,Y 509.483,Z 690.101,A -85,B 0,C 180,E1 -5482.271,E2 -5482.271} C_VEL
LIN {X 0,Y 509.349,Z 696.29,A -85,B 0,C 180,E1 -5483.443,E2 -5483.443} C_VEL
LIN {X 0,Y 509.247,Z 702.101,A -85,B 0,C 180,E1 -5484.854,E2 -5484.854} C_VEL
LIN {X 0,Y 509.296,Z 705.773,A -85,B 0,C 180,E1 -5486.044,E2 -5486.044} C_VEL
LIN {X 0,Y 509.201,Z 707.657,A -85,B 0,C 180,E1 -5486.835,E2 -5486.835} C_VEL
LIN {X 0,Y 509.19,Z 709.073,A -85,B 0,C 180,E1 -5487.627,E2 -5487.627} C_VEL
LIN {X 0,Y 509.089,Z 710.687,A -85,B 0,C 180,E1 -5489.209,E2 -5489.209} C_VEL
LIN {X 0,Y 509.087,Z 710.9,A -85,B 0,C 180,E1 -5490,E2 -5490} C_VEL
LIN {X 0,Y 509.09,Z 710.675,A -85,B 0,C 180,E1 -5490.791,E2 -5490.791} C_VEL
LIN {X 0,Y 509.19,Z 709.041,A -85,B 0,C 180,E1 -5492.373,E2 -5492.373} C_VEL
LIN {X 0,Y 509.214,Z 707.608,A -85,B 0,C 180,E1 -5493.165,E2 -5493.165} C_VEL
LIN {X 0,Y 509.255,Z 704.609,A -85,B 0,C 180,E1 -5494.353,E2 -5494.353} C_VEL
LIN {X 0,Y 509.338,Z 700.551,A -85,B 0,C 180,E1 -5495.543,E2 -5495.543} C_VEL
LIN {X 0,Y 509.404,Z 694.76,A -85,B 0,C 180,E1 -5496.845,E2 -5496.845} C_VEL
LIN {X 0,Y 509.528,Z 687.475,A -85,B 0,C 180,E1 -5498.128,E2 -5498.128} C_VEL
LIN {X 0,Y 509.737,Z 678.994,A -85,B 0,C 180,E1 -5499.324,E2 -5499.324} C_VEL
LIN {X 0,Y 510,Z 670.278,A -85,B 0,C 180,E1 -5500.32,E2 -5500.32} C_VEL
LIN {X 0,Y 510.271,Z 659.527,A -85,B 0,C 180,E1 -5501.319,E2 -5501.319} C_VEL
LIN {X 0,Y 510.564,Z 648.439,A -85,B 0,C 180,E1 -5502.147,E2 -5502.147} C_VEL
LIN {X 0,Y 510.914,Z 636.076,A -85,B 0,C 180,E1 -5502.866,E2 -5502.866} C_VEL
LIN {X 0,Y 511.215,Z 623.539,A -85,B 0,C 180,E1 -5503.415,E2 -5503.415} C_VEL
LIN {X 0,Y 511.472,Z 610.63,A -85,B 0,C 180,E1 -5503.813,E2 -5503.813} C_VEL
LIN {X 0,Y 511.702,Z 595.37,A -85,B 0,C 180,E1 -5504.085,E2 -5504.085} C_VEL
LIN {X 0,Y 512.006,Z 509.117,A -85,B 0,C 180,E1 -5505.334,E2 -5505.334} C_VEL
LIN {X 0,Y 510.307,Z 496.174,A -85,B 0,C 180,E1 -5505.587,E2 -5505.587} C_VEL
LIN {X 0,Y 510.705,Z 476.817,A -85,B 0,C 180,E1 -5508.279,E2 -5508.279} C_VEL
LIN {X 0,Y 511.291,Z 454.926,A -85,B 0,C 180,E1 -5511.362,E2 -5511.362} C_VEL
LIN {X 0,Y 511.833,Z 432.98,A -85,B 0,C 180,E1 -5514.51,E2 -5514.51} C_VEL
LIN {X 0,Y 511.777,Z 429.699,A -85,B 0,C 180,E1 -5514.994,E2 -5514.994} C_VEL
LIN {X 0,Y 509.901,Z 419.972,A -85,B 0,C 180,E1 -5516.533,E2 -5516.533} C_VEL
LIN {X 0,Y 509.88,Z 419.975,A -85,B 0,C 180,E1 -5518.844,E2 -5518.844} C_VEL
LIN {X 0,Y 509.824,Z 419.981,A -85,B 0,C 180,E1 -5521.59,E2 -5521.59} C_VEL
LIN {X 0,Y 509.853,Z 419.977,A -85,B 0,C 180,E1 -5524.414,E2 -5524.414} C_VEL
LIN {X 0,Y 509.82,Z 419.979,A -85,B 0,C 180,E1 -5527.341,E2 -5527.341} C_VEL
LIN {X 0,Y 509.842,Z 419.977,A -85,B 0,C 180,E1 -5530.382,E2 -5530.382} C_VEL
LIN {X 0,Y 509.826,Z 419.979,A -85,B 0,C 180,E1 -5533.062,E2 -5533.062} C_VEL
LIN {X 0,Y 509.826,Z 419.975,A -85,B 0,C 180,E1 -5535.794,E2 -5535.794} C_VEL
LIN {X 0,Y 509.857,Z 419.979,A -85,B 0,C 180,E1 -5538.574,E2 -5538.574} C_VEL
LIN {X 0,Y 509.853,Z 419.971,A -85,B 0,C 180,E1 -5541.787,E2 -5541.787} C_VEL
LIN {X 0,Y 509.83,Z 419.98,A -85,B 0,C 180,E1 -5544.622,E2 -5544.622} C_VEL
LIN {X 0,Y 509.865,Z 419.969,A -85,B 0,C 180,E1 -5547.481,E2 -5547.481} C_VEL
LIN {X 0,Y 509.857,Z 419.977,A -85,B 0,C 180,E1 -5550.275,E2 -5550.275} C_VEL
LIN {X 0,Y 509.825,Z 419.976,A -85,B 0,C 180,E1 -5552.941,E2 -5552.941} C_VEL
LIN {X 0,Y 509.838,Z 419.975,A -85,B 0,C 180,E1 -5555.572,E2 -5555.572} C_VEL
LIN {X 0,Y 509.811,Z 419.983,A -85,B 0,C 180,E1 -5558.148,E2 -5558.148} C_VEL
LIN {X 0,Y 509.81,Z 419.979,A -85,B 0,C 180,E1 -5560.679,E2 -5560.679} C_VEL
LIN {X 0,Y 509.785,Z 419.98,A -85,B 0,C 180,E1 -5563.171,E2 -5563.171} C_VEL
LIN {X 0,Y 509.822,Z 419.98,A -85,B 0,C 180,E1 -5565.633,E2 -5565.633} C_VEL
LIN {X 0,Y 509.892,Z 419.974,A -85,B 0,C 180,E1 -5568.132,E2 -5568.132} C_VEL
LIN {X 0,Y 509.873,Z 419.972,A -85,B 0,C 180,E1 -5571.279,E2 -5571.279} C_VEL
LIN {X 0,Y 509.898,Z 419.974,A -85,B 0,C 180,E1 -5573.669,E2 -5573.669} C_VEL
LIN {X 0,Y 509.888,Z 419.972,A -85,B 0,C 180,E1 -5576.839,E2 -5576.839} C_VEL
LIN {X 0,Y 509.987,Z 419.99,A -85,B 0,C 180,E1 -5578.124,E2 -5578.124} C_VEL
LIN {X 0,Y 510.327,Z 424.504,A -85,B 0,C 180,E1 -5579.211,E2 -5579.211} C_VEL
LIN {X 0,Y 510.323,Z 425.757,A -85,B 0,C 180,E1 -5579.507,E2 -5579.507} C_VEL
LIN {X 0,Y 512.315,Z 435.552,A -85,B 0,C 180,E1 -5579.73,E2 -5579.73} C_VEL
LIN {X 0,Y 511.609,Z 531.543,A -85,B 0,C 180,E1 -5581.156,E2 -5581.156} C_VEL
LIN {X 0,Y 511.428,Z 545.082,A -85,B 0,C 180,E1 -5581.526,E2 -5581.526} C_VEL
LIN {X 0,Y 511.232,Z 557.295,A -85,B 0,C 180,E1 -5582.019,E2 -5582.019} C_VEL
LIN {X 0,Y 510.982,Z 569.032,A -85,B 0,C 180,E1 -5582.661,E2 -5582.661} C_VEL
LIN {X 0,Y 510.589,Z 580.352,A -85,B 0,C 180,E1 -5583.452,E2 -5583.452} C_VEL
LIN {X 0,Y 510.312,Z 590.522,A -85,B 0,C 180,E1 -5584.344,E2 -5584.344} C_VEL
LIN {X 0,Y 510.038,Z 599.679,A -85,B 0,C 180,E1 -5585.337,E2 -5585.337} C_VEL
LIN {X 0,Y 509.785,Z 608.358,A -85,B 0,C 180,E1 -5586.5,E2 -5586.5} C_VEL
LIN {X 0,Y 509.616,Z 615.712,A -85,B 0,C 180,E1 -5587.727,E2 -5587.727} C_VEL
LIN {X 0,Y 509.473,Z 620.56,A -85,B 0,C 180,E1 -5588.728,E2 -5588.728} C_VEL
LIN {X 0,Y 509.367,Z 625.247,A -85,B 0,C 180,E1 -5589.931,E2 -5589.931} C_VEL
LIN {X 0,Y 509.273,Z 628.828,A -85,B 0,C 180,E1 -5591.14,E2 -5591.14} C_VEL
LIN {X 0,Y 509.217,Z 630.657,A -85,B 0,C 180,E1 -5591.948,E2 -5591.948} C_VEL
LIN {X 0,Y 509.168,Z 632.044,A -85,B 0,C 180,E1 -5592.759,E2 -5592.759} C_VEL
LIN {X 0,Y 509.14,Z 632.992,A -85,B 0,C 180,E1 -5593.572,E2 -5593.572} C_VEL
LIN {X 0,Y 509.143,Z 633.665,A -85,B 0,C 180,E1 -5594.926,E2 -5594.926} C_VEL
LIN {X 0,Y 509.125,Z 633.346,A -85,B 0,C 180,E1 -5596.026,E2 -5596.026} C_VEL
LIN {X 0,Y 509.129,Z 632.598,A -85,B 0,C 180,E1 -5596.851,E2 -5596.851} C_VEL
LIN {X 0,Y 509.18,Z 631.29,A -85,B 0,C 180,E1 -5597.752,E2 -5597.752} C_VEL
LIN {X 0,Y 509.224,Z 628.795,A -85,B 0,C 180,E1 -5598.925,E2 -5598.925} C_VEL
LIN {X 0,Y 509.359,Z 624.836,A -85,B 0,C 180,E1 -5600.24,E2 -5600.24} C_VEL
LIN {X 0,Y 509.437,Z 620.039,A -85,B 0,C 180,E1 -5601.444,E2 -5601.444} C_VEL
LIN {X 0,Y 509.608,Z 613.578,A -85,B 0,C 180,E1 -5602.715,E2 -5602.715} C_VEL
LIN {X 0,Y 509.836,Z 605.328,A -85,B 0,C 180,E1 -5603.995,E2 -5603.995} C_VEL
LIN {X 0,Y 510.115,Z 596.627,A -85,B 0,C 180,E1 -5605.076,E2 -5605.076} C_VEL
LIN {X 0,Y 510.393,Z 587.189,A -85,B 0,C 180,E1 -5606.035,E2 -5606.035} C_VEL
LIN {X 0,Y 510.712,Z 576.205,A -85,B 0,C 180,E1 -5606.934,E2 -5606.934} C_VEL
LIN {X 0,Y 511.02,Z 565.013,A -85,B 0,C 180,E1 -5607.656,E2 -5607.656} C_VEL
LIN {X 0,Y 511.319,Z 553.104,A -85,B 0,C 180,E1 -5608.25,E2 -5608.25} C_VEL
LIN {X 0,Y 511.533,Z 540.367,A -85,B 0,C 180,E1 -5608.715,E2 -5608.715} C_VEL
LIN {X 0,Y 511.673,Z 527.509,A -85,B 0,C 180,E1 -5609.014,E2 -5609.014} C_VEL
LIN {X 0,Y 512.165,Z 434.459,A -85,B 0,C 180,E1 -5610.375,E2 -5610.375} C_VEL
LIN {X 0,Y 510.183,Z 424.615,A -85,B 0,C 180,E1 -5610.602,E2 -5610.602} C_VEL
LIN {X 0,Y 509.88,Z 419.975,A -85,B 0,C 180,E1 -5611.673,E2 -5611.673} C_VEL
LIN {X 0,Y 509.837,Z 419.98,A -85,B 0,C 180,E1 -5614.415,E2 -5614.415} C_VEL
LIN {X 0,Y 509.816,Z 419.976,A -85,B 0,C 180,E1 -5615.299,E2 -5615.299} C_VEL
LIN {X 0,Y 509.17,Z 420.06,A -85,B 0,C 180,E1 -5615.959,E2 -5615.959} C_VEL
LIN {X 0,Y 506.301,Z 420.421,A -85,B 0,C 180,E1 -5617.028,E2 -5617.028} C_VEL
LIN {X 0,Y 503.873,Z 420.724,A -85,B 0,C 180,E1 -5617.89,E2 -5617.89} C_VEL
LIN {X 0,Y 502.847,Z 420.849,A -85,B 0,C 180,E1 -5618.556,E2 -5618.556} C_VEL
LIN {X 0,Y 502.774,Z 420.855,A -85,B 0,C 180,E1 -5618.782,E2 -5618.782} C_VEL
LIN {X 0,Y 502.798,Z 420.854,A -85,B 0,C 180,E1 -5622.139,E2 -5622.139} C_VEL
LIN {X 0,Y 502.788,Z 420.85,A -85,B 0,C 180,E1 -5625.47,E2 -5625.47} C_VEL
LIN {X 0,Y 502.773,Z 420.854,A -85,B 0,C 180,E1 -5628.929,E2 -5628.929} C_VEL
LIN {X 0,Y 502.763,Z 420.857,A -85,B 0,C 180,E1 -5632.043,E2 -5632.043} C_VEL
LIN {X 0,Y 502.791,Z 420.851,A -85,B 0,C 180,E1 -5635.033,E2 -5635.033} C_VEL
LIN {X 0,Y 502.785,Z 420.853,A -85,B 0,C 180,E1 -5637.915,E2 -5637.915} C_VEL
LIN {X 0,Y 502.807,Z 420.853,A -85,B 0,C 180,E1 -5640.711,E2 -5640.711} C_VEL
LIN {X 0,Y 502.786,Z 420.85,A -85,B 0,C 180,E1 -5643.457,E2 -5643.457} C_VEL
LIN {X 0,Y 502.77,Z 420.856,A -85,B 0,C 180,E1 -5646.085,E2 -5646.085} C_VEL
LIN {X 0,Y 502.784,Z 420.856,A -85,B 0,C 180,E1 -5648.688,E2 -5648.688} C_VEL
LIN {X 0,Y 502.814,Z 420.847,A -85,B 0,C 180,E1 -5651.247,E2 -5651.247} C_VEL
LIN {X 0,Y 502.837,Z 420.85,A -85,B 0,C 180,E1 -5654.664,E2 -5654.664} C_VEL
LIN {X 0,Y 502.879,Z 420.842,A -85,B 0,C 180,E1 -5658.039,E2 -5658.039} C_VEL
LIN {X 0,Y 502.864,Z 420.842,A -85,B 0,C 180,E1 -5661.156,E2 -5661.156} C_VEL
LIN {X 0,Y 502.918,Z 420.842,A -85,B 0,C 180,E1 -5664.386,E2 -5664.386} C_VEL
LIN {X 0,Y 503.02,Z 420.821,A -85,B 0,C 180,E1 -5667.597,E2 -5667.597} C_VEL
LIN {X 0,Y 503.012,Z 420.827,A -85,B 0,C 180,E1 -5670.8,E2 -5670.8} C_VEL
LIN {X 0,Y 503.019,Z 420.829,A -85,B 0,C 180,E1 -5672.402,E2 -5672.402} C_VEL
LIN {X 0,Y 502.935,Z 420.832,A -85,B 0,C 180,E1 -5675.613,E2 -5675.613} C_VEL
LIN {X 0,Y 502.88,Z 420.841,A -85,B 0,C 180,E1 -5678.033,E2 -5678.033} C_VEL
LIN {X 0,Y 502.877,Z 420.839,A -85,B 0,C 180,E1 -5681.283,E2 -5681.283} C_VEL
LIN {X 0,Y 502.851,Z 420.851,A -85,B 0,C 180,E1 -5684.57,E2 -5684.57} C_VEL
LIN {X 0,Y 502.823,Z 420.847,A -85,B 0,C 180,E1 -5687.908,E2 -5687.908} C_VEL
LIN {X 0,Y 502.83,Z 420.854,A -85,B 0,C 180,E1 -5690.536,E2 -5690.536} C_VEL
LIN {X 0,Y 502.789,Z 420.852,A -85,B 0,C 180,E1 -5693.04,E2 -5693.04} C_VEL
LIN {X 0,Y 502.797,Z 420.849,A -85,B 0,C 180,E1 -5695.678,E2 -5695.678} C_VEL
LIN {X 0,Y 502.796,Z 420.856,A -85,B 0,C 180,E1 -5698.375,E2 -5698.375} C_VEL
LIN {X 0,Y 502.796,Z 420.851,A -85,B 0,C 180,E1 -5701.143,E2 -5701.143} C_VEL
LIN {X 0,Y 502.803,Z 420.85,A -85,B 0,C 180,E1 -5703.994,E2 -5703.994} C_VEL
LIN {X 0,Y 502.764,Z 420.854,A -85,B 0,C 180,E1 -5707.176,E2 -5707.176} C_VEL
LIN {X 0,Y 502.784,Z 420.853,A -85,B 0,C 180,E1 -5710.015,E2 -5710.015} C_VEL
LIN {X 0,Y 502.803,Z 420.852,A -85,B 0,C 180,E1 -5712.199,E2 -5712.199} C_VEL
LIN {X 0,Y 502.785,Z 420.851,A -85,B 0,C 180,E1 -5715.47,E2 -5715.47} C_VEL
LIN {X 0,Y 502.794,Z 420.85,A -85,B 0,C 180,E1 -5717.86,E2 -5717.86} C_VEL
LIN {X 0,Y 502.8,Z 420.852,A -85,B 0,C 180,E1 -5721.024,E2 -5721.024} C_VEL
LIN {X 0,Y 502.77,Z 420.856,A -85,B 0,C 180,E1 -5724.17,E2 -5724.17} C_VEL
LIN {X 0,Y 502.832,Z 420.848,A -85,B 0,C 180,E1 -5726.993,E2 -5726.993} C_VEL
LIN {X 0,Y 502.814,Z 420.849,A -85,B 0,C 180,E1 -5730.065,E2 -5730.065} C_VEL
LIN {X 0,Y 502.823,Z 420.854,A -85,B 0,C 180,E1 -5732.533,E2 -5732.533} C_VEL
LIN {X 0,Y 502.784,Z 420.852,A -85,B 0,C 180,E1 -5735.31,E2 -5735.31} C_VEL
LIN {X 0,Y 502.78,Z 420.852,A -85,B 0,C 180,E1 -5737.826,E2 -5737.826} C_VEL
LIN {X 0,Y 502.823,Z 420.852,A -85,B 0,C 180,E1 -5740.4,E2 -5740.4} C_VEL
LIN {X 0,Y 502.817,Z 420.851,A -85,B 0,C 180,E1 -5742.931,E2 -5742.931} C_VEL
LIN {X 0,Y 502.843,Z 420.844,A -85,B 0,C 180,E1 -5745.429,E2 -5745.429} C_VEL
LIN {X 0,Y 502.877,Z 420.847,A -85,B 0,C 180,E1 -5748.717,E2 -5748.717} C_VEL
LIN {X 0,Y 502.901,Z 420.837,A -85,B 0,C 180,E1 -5751.967,E2 -5751.967} C_VEL
LIN {X 0,Y 502.929,Z 420.838,A -85,B 0,C 180,E1 -5754.386,E2 -5754.386} C_VEL
LIN {X 0,Y 503.024,Z 420.821,A -85,B 0,C 180,E1 -5757.598,E2 -5757.598} C_VEL
LIN {X 0,Y 503.028,Z 420.821,A -85,B 0,C 180,E1 -5760,E2 -5760} C_VEL
LIN {X 0,Y 503.025,Z 420.826,A -85,B 0,C 180,E1 -5762.402,E2 -5762.402} C_VEL
LIN {X 0,Y 502.936,Z 420.832,A -85,B 0,C 180,E1 -5765.614,E2 -5765.614} C_VEL
LIN {X 0,Y 502.901,Z 420.837,A -85,B 0,C 180,E1 -5768.033,E2 -5768.033} C_VEL
LIN {X 0,Y 502.877,Z 420.84,A -85,B 0,C 180,E1 -5771.283,E2 -5771.283} C_VEL
LIN {X 0,Y 502.852,Z 420.85,A -85,B 0,C 180,E1 -5774.571,E2 -5774.571} C_VEL
LIN {X 0,Y 502.823,Z 420.846,A -85,B 0,C 180,E1 -5777.909,E2 -5777.909} C_VEL
LIN {X 0,Y 502.829,Z 420.852,A -85,B 0,C 180,E1 -5780.536,E2 -5780.536} C_VEL
LIN {X 0,Y 502.791,Z 420.854,A -85,B 0,C 180,E1 -5783.041,E2 -5783.041} C_VEL
LIN {X 0,Y 502.811,Z 420.847,A -85,B 0,C 180,E1 -5785.677,E2 -5785.677} C_VEL
LIN {X 0,Y 502.835,Z 420.849,A -85,B 0,C 180,E1 -5788.373,E2 -5788.373} C_VEL
LIN {X 0,Y 502.793,Z 420.85,A -85,B 0,C 180,E1 -5791.499,E2 -5791.499} C_VEL
LIN {X 0,Y 502.804,Z 420.849,A -85,B 0,C 180,E1 -5793.994,E2 -5793.994} C_VEL
LIN {X 0,Y 502.778,Z 420.854,A -85,B 0,C 180,E1 -5797.178,E2 -5797.178} C_VEL
LIN {X 0,Y 502.788,Z 420.851,A -85,B 0,C 180,E1 -5800.015,E2 -5800.015} C_VEL
LIN {X 0,Y 502.803,Z 420.85,A -85,B 0,C 180,E1 -5802.199,E2 -5802.199} C_VEL
LIN {X 0,Y 502.801,Z 420.849,A -85,B 0,C 180,E1 -5805.468,E2 -5805.468} C_VEL
LIN {X 0,Y 502.82,Z 420.852,A -85,B 0,C 180,E1 -5808.934,E2 -5808.934} C_VEL
LIN {X 0,Y 502.791,Z 420.851,A -85,B 0,C 180,E1 -5812.046,E2 -5812.046} C_VEL
LIN {X 0,Y 502.798,Z 420.855,A -85,B 0,C 180,E1 -5815.034,E2 -5815.034} C_VEL
LIN {X 0,Y 502.784,Z 420.851,A -85,B 0,C 180,E1 -5817.916,E2 -5817.916} C_VEL
LIN {X 0,Y 502.824,Z 420.854,A -85,B 0,C 180,E1 -5820.712,E2 -5820.712} C_VEL
LIN {X 0,Y 502.889,Z 421.002,A -85,B 0,C 180,E1 -5823.049,E2 -5823.049} C_VEL
LIN {X 0,Y 505.056,Z 431.578,A -85,B 0,C 180,E1 -5824.756,E2 -5824.756} C_VEL
LIN {X 0,Y 505.06,Z 439.773,A -85,B 0,C 180,E1 -5825.983,E2 -5825.983} C_VEL
LIN {X 0,Y 504.312,Z 461.374,A -85,B 0,C 180,E1 -5829.135,E2 -5829.135} C_VEL
LIN {X 0,Y 503.759,Z 482.108,A -85,B 0,C 180,E1 -5832.126,E2 -5832.126} C_VEL
LIN {X 0,Y 503.363,Z 496.645,A -85,B 0,C 180,E1 -5834.199,E2 -5834.199} C_VEL
LIN {X 0,Y 505.24,Z 510.889,A -85,B 0,C 180,E1 -5834.478,E2 -5834.478} C_VEL
LIN {X 0,Y 504.701,Z 604.927,A -85,B 0,C 180,E1 -5835.87,E2 -5835.87} C_VEL
LIN {X 0,Y 504.469,Z 617.672,A -85,B 0,C 180,E1 -5836.198,E2 -5836.198} C_VEL
LIN {X 0,Y 504.116,Z 630.727,A -85,B 0,C 180,E1 -5836.701,E2 -5836.701} C_VEL
LIN {X 0,Y 503.844,Z 641.952,A -85,B 0,C 180,E1 -5837.288,E2 -5837.288} C_VEL
LIN {X 0,Y 503.526,Z 652.924,A -85,B 0,C 180,E1 -5838.017,E2 -5838.017} C_VEL
LIN {X 0,Y 503.176,Z 663.812,A -85,B 0,C 180,E1 -5838.928,E2 -5838.928} C_VEL
LIN {X 0,Y 502.869,Z 673.618,A -85,B 0,C 180,E1 -5839.939,E2 -5839.939} C_VEL
LIN {X 0,Y 502.61,Z 681.658,A -85,B 0,C 180,E1 -5840.95,E2 -5840.95} C_VEL
LIN {X 0,Y 502.404,Z 689.525,A -85,B 0,C 180,E1 -5842.161,E2 -5842.161} C_VEL
LIN {X 0,Y 502.263,Z 696.205,A -85,B 0,C 180,E1 -5843.455,E2 -5843.455} C_VEL
LIN {X 0,Y 502.184,Z 701.554,A -85,B 0,C 180,E1 -5844.781,E2 -5844.781} C_VEL
LIN {X 0,Y 502.205,Z 705.232,A -85,B 0,C 180,E1 -5845.988,E2 -5845.988} C_VEL
LIN {X 0,Y 502.124,Z 707.121,A -85,B 0,C 180,E1 -5846.791,E2 -5846.791} C_VEL
LIN {X 0,Y 502.121,Z 708.542,A -85,B 0,C 180,E1 -5847.594,E2 -5847.594} C_VEL
LIN {X 0,Y 502.008,Z 710.154,A -85,B 0,C 180,E1 -5849.198,E2 -5849.198} C_VEL
LIN {X 0,Y 502.008,Z 710.365,A -85,B 0,C 180,E1 -5850,E2 -5850} C_VEL
LIN {X 0,Y 502.01,Z 710.137,A -85,B 0,C 180,E1 -5850.802,E2 -5850.802} C_VEL
LIN {X 0,Y 502.122,Z 708.489,A -85,B 0,C 180,E1 -5852.407,E2 -5852.407} C_VEL
LIN {X 0,Y 502.135,Z 707.047,A -85,B 0,C 180,E1 -5853.21,E2 -5853.21} C_VEL
LIN {X 0,Y 502.149,Z 704.03,A -85,B 0,C 180,E1 -5854.415,E2 -5854.415} C_VEL
LIN {X 0,Y 502.251,Z 699.953,A -85,B 0,C 180,E1 -5855.621,E2 -5855.621} C_VEL
LIN {X 0,Y 502.333,Z 693.778,A -85,B 0,C 180,E1 -5857.012,E2 -5857.012} C_VEL
LIN {X 0,Y 502.477,Z 686.818,A -85,B 0,C 180,E1 -5858.243,E2 -5858.243} C_VEL
LIN {X 0,Y 502.688,Z 678.301,A -85,B 0,C 180,E1 -5859.455,E2 -5859.455} C_VEL
LIN {X 0,Y 502.969,Z 669.541,A -85,B 0,C 180,E1 -5860.466,E2 -5860.466} C_VEL
LIN {X 0,Y 503.255,Z 658.738,A -85,B 0,C 180,E1 -5861.479,E2 -5861.479} C_VEL
LIN {X 0,Y 503.58,Z 647.409,A -85,B 0,C 180,E1 -5862.331,E2 -5862.331} C_VEL
LIN {X 0,Y 503.932,Z 635.133,A -85,B 0,C 180,E1 -5863.048,E2 -5863.048} C_VEL
LIN {X 0,Y 504.302,Z 622.499,A -85,B 0,C 180,E1 -5863.602,E2 -5863.602} C_VEL
LIN {X 0,Y 504.542,Z 609.29,A -85,B 0,C 180,E1 -5864.006,E2 -5864.006} C_VEL
LIN {X 0,Y 504.792,Z 593.658,A -85,B 0,C 180,E1 -5864.282,E2 -5864.282} C_VEL
LIN {X 0,Y 505.132,Z 509.63,A -85,B 0,C 180,E1 -5865.529,E2 -5865.529} C_VEL
LIN {X 0,Y 503.273,Z 495.393,A -85,B 0,C 180,E1 -5865.827,E2 -5865.827} C_VEL
LIN {X 0,Y 503.712,Z 476.446,A -85,B 0,C 180,E1 -5868.506,E2 -5868.506} C_VEL
LIN {X 0,Y 504.34,Z 454.321,A -85,B 0,C 180,E1 -5871.672,E2 -5871.672} C_VEL
LIN {X 0,Y 504.942,Z 432.554,A -85,B 0,C 180,E1 -5874.856,E2 -5874.856} C_VEL
LIN {X 0,Y 503.382,Z 423.347,A -85,B 0,C 180,E1 -5876.314,E2 -5876.314} C_VEL
LIN {X 0,Y 502.861,Z 420.85,A -85,B 0,C 180,E1 -5876.743,E2 -5876.743} C_VEL
LIN {X 0,Y 502.828,Z 420.853,A -85,B 0,C 180,E1 -5879.288,E2 -5879.288} C_VEL
LIN {X 0,Y 502.787,Z 420.857,A -85,B 0,C 180,E1 -5882.085,E2 -5882.085} C_VEL
LIN {X 0,Y 502.805,Z 420.86,A -85,B 0,C 180,E1 -5884.966,E2 -5884.966} C_VEL
LIN {X 0,Y 502.797,Z 420.852,A -85,B 0,C 180,E1 -5887.954,E2 -5887.954} C_VEL
LIN {X 0,Y 502.823,Z 420.853,A -85,B 0,C 180,E1 -5891.066,E2 -5891.066} C_VEL
LIN {X 0,Y 502.79,Z 420.857,A -85,B 0,C 180,E1 -5894.53,E2 -5894.53} C_VEL
LIN {X 0,Y 502.798,Z 420.85,A -85,B 0,C 180,E1 -5897.861,E2 -5897.861} C_VEL
LIN {X 0,Y 502.804,Z 420.852,A -85,B 0,C 180,E1 -5901.024,E2 -5901.024} C_VEL
LIN {X 0,Y 502.774,Z 420.856,A -85,B 0,C 180,E1 -5904.17,E2 -5904.17} C_VEL
LIN {X 0,Y 502.837,Z 420.846,A -85,B 0,C 180,E1 -5906.994,E2 -5906.994} C_VEL
LIN {X 0,Y 502.814,Z 420.852,A -85,B 0,C 180,E1 -5910.066,E2 -5910.066} C_VEL
LIN {X 0,Y 502.787,Z 420.852,A -85,B 0,C 180,E1 -5913.429,E2 -5913.429} C_VEL
LIN {X 0,Y 502.77,Z 420.859,A -85,B 0,C 180,E1 -5916.085,E2 -5916.085} C_VEL
LIN {X 0,Y 502.764,Z 420.857,A -85,B 0,C 180,E1 -5918.688,E2 -5918.688} C_VEL
LIN {X 0,Y 502.787,Z 420.857,A -85,B 0,C 180,E1 -5921.9,E2 -5921.9} C_VEL
LIN {X 0,Y 502.795,Z 420.853,A -85,B 0,C 180,E1 -5924.683,E2 -5924.683} C_VEL
LIN {X 0,Y 502.843,Z 420.852,A -85,B 0,C 180,E1 -5928.06,E2 -5928.06} C_VEL
LIN {X 0,Y 502.837,Z 420.848,A -85,B 0,C 180,E1 -5931.156,E2 -5931.156} C_VEL
LIN {X 0,Y 502.851,Z 420.851,A -85,B 0,C 180,E1 -5933.58,E2 -5933.58} C_VEL
LIN {X 0,Y 502.745,Z 420.865,A -85,B 0,C 180,E1 -5935.992,E2 -5935.992} C_VEL
LIN {X 0,Y 502.987,Z 420.859,A -85,B 0,C 180,E1 -5937.948,E2 -5937.948} C_VEL
LIN {X 0,Y 503.385,Z 426.012,A -85,B 0,C 180,E1 -5939.2,E2 -5939.2} C_VEL
LIN {X 0,Y 503.374,Z 426.508,A -85,B 0,C 180,E1 -5939.3,E2 -5939.3} C_VEL
LIN {X 0,Y 505.469,Z 436.489,A -85,B 0,C 180,E1 -5939.527,E2 -5939.527} C_VEL
LIN {X 0,Y 504.711,Z 531.807,A -85,B 0,C 180,E1 -5940.972,E2 -5940.972} C_VEL
LIN {X 0,Y 504.532,Z 545.424,A -85,B 0,C 180,E1 -5941.347,E2 -5941.347} C_VEL
LIN {X 0,Y 504.329,Z 557.698,A -85,B 0,C 180,E1 -5941.847,E2 -5941.847} C_VEL
LIN {X 0,Y 504.059,Z 569.486,A -85,B 0,C 180,E1 -5942.497,E2 -5942.497} C_VEL
LIN {X 0,Y 503.634,Z 580.838,A -85,B 0,C 180,E1 -5943.3,E2 -5943.3} C_VEL
LIN {X 0,Y 503.34,Z 591.034,A -85,B 0,C 180,E1 -5944.204,E2 -5944.204} C_VEL
LIN {X 0,Y 503.043,Z 600.207,A -85,B 0,C 180,E1 -5945.21,E2 -5945.21} C_VEL
LIN {X 0,Y 502.76,Z 609.107,A -85,B 0,C 180,E1 -5946.421,E2 -5946.421} C_VEL
LIN {X 0,Y 502.59,Z 616.272,A -85,B 0,C 180,E1 -5947.634,E2 -5947.634} C_VEL
LIN {X 0,Y 502.4,Z 622.005,A -85,B 0,C 180,E1 -5948.852,E2 -5948.852} C_VEL
LIN {X 0,Y 502.313,Z 626.498,A -85,B 0,C 180,E1 -5950.072,E2 -5950.072} C_VEL
LIN {X 0,Y 502.212,Z 630.556,A -85,B 0,C 180,E1 -5951.595,E2 -5951.595} C_VEL
LIN {X 0,Y 502.1,Z 632.874,A -85,B 0,C 180,E1 -5952.941,E2 -5952.941} C_VEL
LIN {X 0,Y 502.063,Z 633.74,A -85,B 0,C 180,E1 -5953.767,E2 -5953.767} C_VEL
LIN {X 0,Y 502.076,Z 634.217,A -85,B 0,C 180,E1 -5955.014,E2 -5955.014} C_VEL
LIN {X 0,Y 502.042,Z 633.741,A -85,B 0,C 180,E1 -5956.259,E2 -5956.259} C_VEL
LIN {X 0,Y 502.057,Z 632.881,A -85,B 0,C 180,E1 -5957.096,E2 -5957.096} C_VEL
LIN {X 0,Y 502.128,Z 631.557,A -85,B 0,C 180,E1 -5957.934,E2 -5957.934} C_VEL
LIN {X 0,Y 502.175,Z 628.729,A -85,B 0,C 180,E1 -5959.201,E2 -5959.201} C_VEL
LIN {X 0,Y 502.319,Z 624.758,A -85,B 0,C 180,E1 -5960.474,E2 -5960.474} C_VEL
LIN {X 0,Y 502.43,Z 619.5,A -85,B 0,C 180,E1 -5961.758,E2 -5961.758} C_VEL
LIN {X 0,Y 502.612,Z 612.724,A -85,B 0,C 180,E1 -5963.049,E2 -5963.049} C_VEL
LIN {X 0,Y 502.92,Z 604.088,A -85,B 0,C 180,E1 -5964.346,E2 -5964.346} C_VEL
LIN {X 0,Y 503.214,Z 595.099,A -85,B 0,C 180,E1 -5965.433,E2 -5965.433} C_VEL
LIN {X 0,Y 503.51,Z 584.986,A -85,B 0,C 180,E1 -5966.418,E2 -5966.418} C_VEL
LIN {X 0,Y 503.888,Z 573.59,A -85,B 0,C 180,E1 -5967.306,E2 -5967.306} C_VEL
LIN {X 0,Y 504.218,Z 562.172,A -85,B 0,C 180,E1 -5968.005,E2 -5968.005} C_VEL
LIN {X 0,Y 504.473,Z 550.587,A -85,B 0,C 180,E1 -5968.546,E2 -5968.546} C_VEL
LIN {X 0,Y 504.697,Z 537.942,A -85,B 0,C 180,E1 -5968.971,E2 -5968.971} C_VEL
LIN {X 0,Y 504.822,Z 524.985,A -85,B 0,C 180,E1 -5969.246,E2 -5969.246} C_VEL
LIN {X 0,Y 505.361,Z 435.241,A -85,B 0,C 180,E1 -5970.581,E2 -5970.581} C_VEL
LIN {X 0,Y 503.218,Z 425.021,A -85,B 0,C 180,E1 -5970.82,E2 -5970.82} C_VEL
LIN {X 0,Y 502.855,Z 420.85,A -85,B 0,C 180,E1 -5971.811,E2 -5971.811} C_VEL
LIN {X 0,Y 502.791,Z 420.853,A -85,B 0,C 180,E1 -5974.967,E2 -5974.967} C_VEL
LIN {X 0,Y 502.767,Z 420.861,A -85,B 0,C 180,E1 -5978.481,E2 -5978.481} C_VEL
LIN {X 0,Y 502.774,Z 420.855,A -85,B 0,C 180,E1 -5978.782,E2 -5978.782} C_VEL
LIN {X 0,Y 502.133,Z 420.933,A -85,B 0,C 180,E1 -5979.45,E2 -5979.45} C_VEL
LIN {X 0,Y 499.279,Z 421.294,A -85,B 0,C 180,E1 -5980.536,E2 -5980.536} C_VEL
LIN {X 0,Y 496.848,Z 421.594,A -85,B 0,C 180,E1 -5981.411,E2 -5981.411} C_VEL
LIN {X 0,Y 495.801,Z 421.725,A -85,B 0,C 180,E1 -5982.086,E2 -5982.086} C_VEL
LIN {X 0,Y 495.716,Z 421.736,A -85,B 0,C 180,E1 -5982.315,E2 -5982.315} C_VEL
LIN {X 0,Y 495.74,Z 421.729,A -85,B 0,C 180,E1 -5985.141,E2 -5985.141} C_VEL
LIN {X 0,Y 495.727,Z 421.736,A -85,B 0,C 180,E1 -5988.215,E2 -5988.215} C_VEL
LIN {X 0,Y 495.743,Z 421.728,A -85,B 0,C 180,E1 -5991.235,E2 -5991.235} C_VEL
LIN {X 0,Y 495.738,Z 421.737,A -85,B 0,C 180,E1 -5994.461,E2 -5994.461} C_VEL
LIN {X 0,Y 495.77,Z 421.724,A -85,B 0,C 180,E1 -5997.405,E2 -5997.405} C_VEL
LIN {X 0,Y 495.76,Z 421.732,A -85,B 0,C 180,E1 -6000.253,E2 -6000.253} C_VEL
LIN {X 0,Y 495.744,Z 421.728,A -85,B 0,C 180,E1 -6003.269,E2 -6003.269} C_VEL
LIN {X 0,Y 495.741,Z 421.734,A -85,B 0,C 180,E1 -6006.612,E2 -6006.612} C_VEL
LIN {X 0,Y 495.781,Z 421.723,A -85,B 0,C 180,E1 -6009.324,E2 -6009.324} C_VEL
LIN {X 0,Y 495.781,Z 421.724,A -85,B 0,C 180,E1 -6011.828,E2 -6011.828} C_VEL
LIN {X 0,Y 495.782,Z 421.723,A -85,B 0,C 180,E1 -6015.217,E2 -6015.217} C_VEL
LIN {X 0,Y 495.853,Z 421.722,A -85,B 0,C 180,E1 -6018.555,E2 -6018.555} C_VEL
LIN {X 0,Y 495.832,Z 421.718,A -85,B 0,C 180,E1 -6021.851,E2 -6021.851} C_VEL
LIN {X 0,Y 495.833,Z 421.718,A -85,B 0,C 180,E1 -6025.121,E2 -6025.121} C_VEL
LIN {X 0,Y 495.988,Z 421.697,A -85,B 0,C 180,E1 -6027.563,E2 -6027.563} C_VEL
LIN {X 0,Y 495.963,Z 421.705,A -85,B 0,C 180,E1 -6030.812,E2 -6030.812} C_VEL
LIN {X 0,Y 495.986,Z 421.706,A -85,B 0,C 180,E1 -6032.436,E2 -6032.436} C_VEL
LIN {X 0,Y 495.893,Z 421.709,A -85,B 0,C 180,E1 -6035.693,E2 -6035.693} C_VEL
LIN {X 0,Y 495.836,Z 421.72,A -85,B 0,C 180,E1 -6038.148,E2 -6038.148} C_VEL
LIN {X 0,Y 495.852,Z 421.714,A -85,B 0,C 180,E1 -6041.445,E2 -6041.445} C_VEL
LIN {X 0,Y 495.795,Z 421.726,A -85,B 0,C 180,E1 -6044.782,E2 -6044.782} C_VEL
LIN {X 0,Y 495.764,Z 421.726,A -85,B 0,C 180,E1 -6047.319,E2 -6047.319} C_VEL
LIN {X 0,Y 495.771,Z 421.726,A -85,B 0,C 180,E1 -6049.89,E2 -6049.89} C_VEL
LIN {X 0,Y 495.76,Z 421.73,A -85,B 0,C 180,E1 -6052.86,E2 -6052.86} C_VEL
LIN {X 0,Y 495.759,Z 421.729,A -85,B 0,C 180,E1 -6056.069,E2 -6056.069} C_VEL
LIN {X 0,Y 495.744,Z 421.733,A -85,B 0,C 180,E1 -6058.816,E2 -6058.816} C_VEL
LIN {X 0,Y 495.755,Z 421.727,A -85,B 0,C 180,E1 -6061.725,E2 -6061.725} C_VEL
LIN {X 0,Y 495.768,Z 421.732,A -85,B 0,C 180,E1 -6064.693,E2 -6064.693} C_VEL
LIN {X 0,Y 495.721,Z 421.731,A -85,B 0,C 180,E1 -6067.562,E2 -6067.562} C_VEL
LIN {X 0,Y 495.755,Z 421.728,A -85,B 0,C 180,E1 -6070.046,E2 -6070.046} C_VEL
LIN {X 0,Y 495.714,Z 421.736,A -85,B 0,C 180,E1 -6072.884,E2 -6072.884} C_VEL
LIN {X 0,Y 495.724,Z 421.732,A -85,B 0,C 180,E1 -6075.998,E2 -6075.998} C_VEL
LIN {X 0,Y 495.739,Z 421.735,A -85,B 0,C 180,E1 -6078.709,E2 -6078.709} C_VEL
LIN {X 0,Y 495.748,Z 421.727,A -85,B 0,C 180,E1 -6081.408,E2 -6081.408} C_VEL
LIN {X 0,Y 495.745,Z 421.735,A -85,B 0,C 180,E1 -6084.462,E2 -6084.462} C_VEL
LIN {X 0,Y 495.767,Z 421.725,A -85,B 0,C 180,E1 -6087.406,E2 -6087.406} C_VEL
LIN {X 0,Y 495.765,Z 421.729,A -85,B 0,C 180,E1 -6090.254,E2 -6090.254} C_VEL
LIN {X 0,Y 495.805,Z 421.721,A -85,B 0,C 180,E1 -6093.255,E2 -6093.255} C_VEL
LIN {X 0,Y 495.742,Z 421.737,A -85,B 0,C 180,E1 -6096.612,E2 -6096.612} C_VEL
LIN {X 0,Y 495.778,Z 421.724,A -85,B 0,C 180,E1 -6099.324,E2 -6099.324} C_VEL
LIN {X 0,Y 495.781,Z 421.723,A -85,B 0,C 180,E1 -6101.828,E2 -6101.828} C_VEL
LIN {X 0,Y 495.824,Z 421.726,A -85,B 0,C 180,E1 -6104.548,E2 -6104.548} C_VEL
LIN {X 0,Y 495.828,Z 421.718,A -85,B 0,C 180,E1 -6107.965,E2 -6107.965} C_VEL
LIN {X 0,Y 495.838,Z 421.719,A -85,B 0,C 180,E1 -6111.03,E2 -6111.03} C_VEL
LIN {X 0,Y 495.884,Z 421.714,A -85,B 0,C 180,E1 -6114.306,E2 -6114.306} C_VEL
LIN {X 0,Y 495.992,Z 421.697,A -85,B 0,C 180,E1 -6117.564,E2 -6117.564} C_VEL
LIN {X 0,Y 495.983,Z 421.705,A -85,B 0,C 180,E1 -6120.812,E2 -6120.812} C_VEL
LIN {X 0,Y 495.993,Z 421.702,A -85,B 0,C 180,E1 -6122.436,E2 -6122.436} C_VEL
LIN {X 0,Y 495.894,Z 421.709,A -85,B 0,C 180,E1 -6125.694,E2 -6125.694} C_VEL
LIN {X 0,Y 495.872,Z 421.714,A -85,B 0,C 180,E1 -6128.148,E2 -6128.148} C_VEL
LIN {X 0,Y 495.852,Z 421.715,A -85,B 0,C 180,E1 -6131.445,E2 -6131.445} C_VEL
LIN {X 0,Y 495.795,Z 421.729,A -85,B 0,C 180,E1 -6134.783,E2 -6134.783} C_VEL
LIN {X 0,Y 495.765,Z 421.726,A -85,B 0,C 180,E1 -6137.319,E2 -6137.319} C_VEL
LIN {X 0,Y 495.771,Z 421.725,A -85,B 0,C 180,E1 -6139.891,E2 -6139.891} C_VEL
LIN {X 0,Y 495.76,Z 421.732,A -85,B 0,C 180,E1 -6142.861,E2 -6142.861} C_VEL
LIN {X 0,Y 495.767,Z 421.726,A -85,B 0,C 180,E1 -6146.069,E2 -6146.069} C_VEL
LIN {X 0,Y 495.769,Z 421.732,A -85,B 0,C 180,E1 -6148.815,E2 -6148.815} C_VEL
LIN {X 0,Y 495.755,Z 421.726,A -85,B 0,C 180,E1 -6151.725,E2 -6151.725} C_VEL
LIN {X 0,Y 495.769,Z 421.734,A -85,B 0,C 180,E1 -6154.694,E2 -6154.694} C_VEL
LIN {X 0,Y 495.729,Z 421.73,A -85,B 0,C 180,E1 -6157.562,E2 -6157.562} C_VEL
LIN {X 0,Y 495.766,Z 421.734,A -85,B 0,C 180,E1 -6160.7,E2 -6160.7} C_VEL
LIN {X 0,Y 495.734,Z 421.73,A -85,B 0,C 180,E1 -6164.001,E2 -6164.001} C_VEL
LIN {X 0,Y 495.727,Z 421.733,A -85,B 0,C 180,E1 -6167.117,E2 -6167.117} C_VEL
LIN {X 0,Y 495.759,Z 421.726,A -85,B 0,C 180,E1 -6169.953,E2 -6169.953} C_VEL
LIN {X 0,Y 495.72,Z 421.737,A -85,B 0,C 180,E1 -6172.555,E2 -6172.555} C_VEL
LIN {X 0,Y 495.778,Z 421.724,A -85,B 0,C 180,E1 -6175.457,E2 -6175.457} C_VEL
LIN {X 0,Y 495.756,Z 421.73,A -85,B 0,C 180,E1 -6178.364,E2 -6178.364} C_VEL
LIN {X 0,Y 495.787,Z 421.728,A -85,B 0,C 180,E1 -6181.508,E2 -6181.508} C_VEL
LIN {X 0,Y 495.831,Z 421.808,A -85,B 0,C 180,E1 -6182.828,E2 -6182.828} C_VEL
LIN {X 0,Y 498.177,Z 433.351,A -85,B 0,C 180,E1 -6184.717,E2 -6184.717} C_VEL
LIN {X 0,Y 498.073,Z 443.59,A -85,B 0,C 180,E1 -6186.267,E2 -6186.267} C_VEL
LIN {X 0,Y 497.265,Z 464.15,A -85,B 0,C 180,E1 -6189.309,E2 -6189.309} C_VEL
LIN {X 0,Y 496.685,Z 484.538,A -85,B 0,C 180,E1 -6192.289,E2 -6192.289} C_VEL
LIN {X 0,Y 496.331,Z 496.155,A -85,B 0,C 180,E1 -6193.969,E2 -6193.969} C_VEL
LIN {X 0,Y 498.416,Z 511.949,A -85,B 0,C 180,E1 -6194.284,E2 -6194.284} C_VEL
LIN {X 0,Y 497.77,Z 605.049,A -85,B 0,C 180,E1 -6195.695,E2 -6195.695} C_VEL
LIN {X 0,Y 497.541,Z 617.541,A -85,B 0,C 180,E1 -6196.028,E2 -6196.028} C_VEL
LIN {X 0,Y 497.148,Z 631.052,A -85,B 0,C 180,E1 -6196.564,E2 -6196.564} C_VEL
LIN {X 0,Y 496.8,Z 643.704,A -85,B 0,C 180,E1 -6197.26,E2 -6197.26} C_VEL
LIN {X 0,Y 496.438,Z 654.854,A -85,B 0,C 180,E1 -6198.051,E2 -6198.051} C_VEL
LIN {X 0,Y 496.071,Z 665.327,A -85,B 0,C 180,E1 -6198.974,E2 -6198.974} C_VEL
LIN {X 0,Y 495.758,Z 674.742,A -85,B 0,C 180,E1 -6200,E2 -6200} C_VEL
LIN {X 0,Y 495.464,Z 683.865,A -85,B 0,C 180,E1 -6201.229,E2 -6201.229} C_VEL
LIN {X 0,Y 495.282,Z 691.219,A -85,B 0,C 180,E1 -6202.458,E2 -6202.458} C_VEL
LIN {X 0,Y 495.131,Z 697.375,A -85,B 0,C 180,E1 -6203.753,E2 -6203.753} C_VEL
LIN {X 0,Y 495.039,Z 702.346,A -85,B 0,C 180,E1 -6205.114,E2 -6205.114} C_VEL
LIN {X 0,Y 495.099,Z 704.691,A -85,B 0,C 180,E1 -6205.93,E2 -6205.93} C_VEL
LIN {X 0,Y 495.048,Z 706.586,A -85,B 0,C 180,E1 -6206.745,E2 -6206.745} C_VEL
LIN {X 0,Y 495.054,Z 708.01,A -85,B 0,C 180,E1 -6207.559,E2 -6207.559} C_VEL
LIN {X 0,Y 494.928,Z 709.62,A -85,B 0,C 180,E1 -6209.187,E2 -6209.187} C_VEL
LIN {X 0,Y 494.929,Z 709.83,A -85,B 0,C 180,E1 -6210,E2 -6210} C_VEL
LIN {X 0,Y 494.93,Z 709.598,A -85,B 0,C 180,E1 -6210.814,E2 -6210.814} C_VEL
LIN {X 0,Y 494.965,Z 708.968,A -85,B 0,C 180,E1 -6211.628,E2 -6211.628} C_VEL
LIN {X 0,Y 495.055,Z 707.937,A -85,B 0,C 180,E1 -6212.441,E2 -6212.441} C_VEL
LIN {X 0,Y 495.06,Z 706.486,A -85,B 0,C 180,E1 -6213.256,E2 -6213.256} C_VEL
LIN {X 0,Y 495.049,Z 703.451,A -85,B 0,C 180,E1 -6214.479,E2 -6214.479} C_VEL
LIN {X 0,Y 495.149,Z 698.252,A -85,B 0,C 180,E1 -6215.979,E2 -6215.979} C_VEL
LIN {X 0,Y 495.27,Z 692.006,A -85,B 0,C 180,E1 -6217.338,E2 -6217.338} C_VEL
LIN {X 0,Y 495.451,Z 684.882,A -85,B 0,C 180,E1 -6218.566,E2 -6218.566} C_VEL
LIN {X 0,Y 495.659,Z 675.951,A -85,B 0,C 180,E1 -6219.797,E2 -6219.797} C_VEL
LIN {X 0,Y 496.017,Z 665.805,A -85,B 0,C 180,E1 -6220.924,E2 -6220.924} C_VEL
LIN {X 0,Y 496.358,Z 655.488,A -85,B 0,C 180,E1 -6221.848,E2 -6221.848} C_VEL
LIN {X 0,Y 496.683,Z 644.034,A -85,B 0,C 180,E1 -6222.669,E2 -6222.669} C_VEL
LIN {X 0,Y 497.067,Z 632.181,A -85,B 0,C 180,E1 -6223.335,E2 -6223.335} C_VEL
LIN {X 0,Y 497.408,Z 619.307,A -85,B 0,C 180,E1 -6223.872,E2 -6223.872} C_VEL
LIN {X 0,Y 497.715,Z 605.686,A -85,B 0,C 180,E1 -6224.255,E2 -6224.255} C_VEL
LIN {X 0,Y 498.112,Z 562.576,A -85,B 0,C 180,E1 -6224.922,E2 -6224.922} C_VEL
LIN {X 0,Y 498.163,Z 509.627,A -85,B 0,C 180,E1 -6225.741,E2 -6225.741} C_VEL
LIN {X 0,Y 496.251,Z 494.835,A -85,B 0,C 180,E1 -6226.045,E2 -6226.045} C_VEL
LIN {X 0,Y 496.796,Z 474.356,A -85,B 0,C 180,E1 -6228.989,E2 -6228.989} C_VEL
LIN {X 0,Y 497.347,Z 453.766,A -85,B 0,C 180,E1 -6231.992,E2 -6231.992} C_VEL
LIN {X 0,Y 498.01,Z 434.716,A -85,B 0,C 180,E1 -6234.825,E2 -6234.825} C_VEL
LIN {X 0,Y 497.201,Z 428.571,A -85,B 0,C 180,E1 -6235.803,E2 -6235.803} C_VEL
LIN {X 0,Y 495.824,Z 421.726,A -85,B 0,C 180,E1 -6236.936,E2 -6236.936} C_VEL
LIN {X 0,Y 495.769,Z 421.73,A -85,B 0,C 180,E1 -6240.147,E2 -6240.147} C_VEL
LIN {X 0,Y 495.797,Z 421.732,A -85,B 0,C 180,E1 -6243.245,E2 -6243.245} C_VEL
LIN {X 0,Y 495.724,Z 421.735,A -85,B 0,C 180,E1 -6246.089,E2 -6246.089} C_VEL
LIN {X 0,Y 495.767,Z 421.734,A -85,B 0,C 180,E1 -6248.768,E2 -6248.768} C_VEL
LIN {X 0,Y 495.76,Z 421.728,A -85,B 0,C 180,E1 -6251.781,E2 -6251.781} C_VEL
LIN {X 0,Y 495.741,Z 421.732,A -85,B 0,C 180,E1 -6255.141,E2 -6255.141} C_VEL
LIN {X 0,Y 495.754,Z 421.73,A -85,B 0,C 180,E1 -6258.218,E2 -6258.218} C_VEL
LIN {X 0,Y 495.753,Z 421.728,A -85,B 0,C 180,E1 -6261.408,E2 -6261.408} C_VEL
LIN {X 0,Y 495.748,Z 421.736,A -85,B 0,C 180,E1 -6264.462,E2 -6264.462} C_VEL
LIN {X 0,Y 495.771,Z 421.725,A -85,B 0,C 180,E1 -6267.406,E2 -6267.406} C_VEL
LIN {X 0,Y 495.761,Z 421.732,A -85,B 0,C 180,E1 -6270.253,E2 -6270.253} C_VEL
LIN {X 0,Y 495.742,Z 421.73,A -85,B 0,C 180,E1 -6273.271,E2 -6273.271} C_VEL
LIN {X 0,Y 495.742,Z 421.733,A -85,B 0,C 180,E1 -6276.612,E2 -6276.612} C_VEL
LIN {X 0,Y 495.728,Z 421.732,A -85,B 0,C 180,E1 -6279.341,E2 -6279.341} C_VEL
LIN {X 0,Y 495.737,Z 421.734,A -85,B 0,C 180,E1 -6281.827,E2 -6281.827} C_VEL
LIN {X 0,Y 495.749,Z 421.73,A -85,B 0,C 180,E1 -6285.216,E2 -6285.216} C_VEL
LIN {X 0,Y 495.815,Z 421.724,A -85,B 0,C 180,E1 -6288.554,E2 -6288.554} C_VEL
LIN {X 0,Y 495.813,Z 421.729,A -85,B 0,C 180,E1 -6291.851,E2 -6291.851} C_VEL
LIN {X 0,Y 495.846,Z 421.722,A -85,B 0,C 180,E1 -6294.306,E2 -6294.306} C_VEL
LIN {X 0,Y 495.966,Z 421.775,A -85,B 0,C 180,E1 -6297.767,E2 -6297.767} C_VEL
LIN {X 0,Y 496.477,Z 427.152,A -85,B 0,C 180,E1 -6299.075,E2 -6299.075} C_VEL
LIN {X 0,Y 498.57,Z 436.32,A -85,B 0,C 180,E1 -6299.293,E2 -6299.293} C_VEL
LIN {X 0,Y 497.826,Z 533.247,A -85,B 0,C 180,E1 -6300.809,E2 -6300.809} C_VEL
LIN {X 0,Y 497.641,Z 546.551,A -85,B 0,C 180,E1 -6301.188,E2 -6301.188} C_VEL
LIN {X 0,Y 497.427,Z 559.144,A -85,B 0,C 180,E1 -6301.72,E2 -6301.72} C_VEL
LIN {X 0,Y 497.116,Z 571.495,A -85,B 0,C 180,E1 -6302.431,E2 -6302.431} C_VEL
LIN {X 0,Y 496.657,Z 582.594,A -85,B 0,C 180,E1 -6303.245,E2 -6303.245} C_VEL
LIN {X 0,Y 496.383,Z 591.535,A -85,B 0,C 180,E1 -6304.059,E2 -6304.059} C_VEL
LIN {X 0,Y 496.052,Z 600.734,A -85,B 0,C 180,E1 -6305.08,E2 -6305.08} C_VEL
LIN {X 0,Y 495.765,Z 609.642,A -85,B 0,C 180,E1 -6306.307,E2 -6306.307} C_VEL
LIN {X 0,Y 495.583,Z 616.816,A -85,B 0,C 180,E1 -6307.538,E2 -6307.538} C_VEL
LIN {X 0,Y 495.403,Z 621.669,A -85,B 0,C 180,E1 -6308.566,E2 -6308.566} C_VEL
LIN {X 0,Y 495.25,Z 626.377,A -85,B 0,C 180,E1 -6309.805,E2 -6309.805} C_VEL
LIN {X 0,Y 495.156,Z 629.961,A -85,B 0,C 180,E1 -6311.047,E2 -6311.047} C_VEL
LIN {X 0,Y 495.069,Z 632.517,A -85,B 0,C 180,E1 -6312.295,E2 -6312.295} C_VEL
LIN {X 0,Y 495.009,Z 633.697,A -85,B 0,C 180,E1 -6313.13,E2 -6313.13} C_VEL
LIN {X 0,Y 494.994,Z 634.411,A -85,B 0,C 180,E1 -6313.967,E2 -6313.967} C_VEL
LIN {X 0,Y 494.994,Z 634.753,A -85,B 0,C 180,E1 -6315.098,E2 -6315.098} C_VEL
LIN {X 0,Y 494.967,Z 634.081,A -85,B 0,C 180,E1 -6316.498,E2 -6316.498} C_VEL
LIN {X 0,Y 495.061,Z 632.07,A -85,B 0,C 180,E1 -6317.982,E2 -6317.982} C_VEL
LIN {X 0,Y 495.14,Z 628.647,A -85,B 0,C 180,E1 -6319.485,E2 -6319.485} C_VEL
LIN {X 0,Y 495.282,Z 624.445,A -85,B 0,C 180,E1 -6320.778,E2 -6320.778} C_VEL
LIN {X 0,Y 495.416,Z 618.888,A -85,B 0,C 180,E1 -6322.082,E2 -6322.082} C_VEL
LIN {X 0,Y 495.65,Z 611.784,A -85,B 0,C 180,E1 -6323.392,E2 -6323.392} C_VEL
LIN {X 0,Y 495.966,Z 603.313,A -85,B 0,C 180,E1 -6324.639,E2 -6324.639} C_VEL
LIN {X 0,Y 496.258,Z 594.316,A -85,B 0,C 180,E1 -6325.703,E2 -6325.703} C_VEL
LIN {X 0,Y 496.613,Z 583.923,A -85,B 0,C 180,E1 -6326.7,E2 -6326.7} C_VEL
LIN {X 0,Y 497.004,Z 572.636,A -85,B 0,C 180,E1 -6327.565,E2 -6327.565} C_VEL
LIN {X 0,Y 497.322,Z 561.072,A -85,B 0,C 180,E1 -6328.256,E2 -6328.256} C_VEL
LIN {X 0,Y 497.641,Z 548.197,A -85,B 0,C 180,E1 -6328.836,E2 -6328.836} C_VEL
LIN {X 0,Y 497.842,Z 535.484,A -85,B 0,C 180,E1 -6329.232,E2 -6329.232} C_VEL
LIN {X 0,Y 497.962,Z 519.965,A -85,B 0,C 180,E1 -6329.515,E2 -6329.515} C_VEL
LIN {X 0,Y 498.565,Z 436.453,A -85,B 0,C 180,E1 -6330.785,E2 -6330.785} C_VEL
LIN {X 0,Y 496.258,Z 425.414,A -85,B 0,C 180,E1 -6331.048,E2 -6331.048} C_VEL
LIN {X 0,Y 495.803,Z 421.729,A -85,B 0,C 180,E1 -6331.957,E2 -6331.957} C_VEL
LIN {X 0,Y 495.76,Z 421.731,A -85,B 0,C 180,E1 -6334.692,E2 -6334.692} C_VEL
LIN {X 0,Y 495.709,Z 421.732,A -85,B 0,C 180,E1 -6337.563,E2 -6337.563} C_VEL
LIN {X 0,Y 495.746,Z 421.731,A -85,B 0,C 180,E1 -6340.045,E2 -6340.045} C_VEL
LIN {X 0,Y 495.716,Z 421.736,A -85,B 0,C 180,E1 -6342.315,E2 -6342.315} C_VEL
LIN {X 0,Y 495.046,Z 421.824,A -85,B 0,C 180,E1 -6342.994,E2 -6342.994} C_VEL
LIN {X 0,Y 492.187,Z 422.176,A -85,B 0,C 180,E1 -6344.095,E2 -6344.095} C_VEL
LIN {X 0,Y 489.781,Z 422.472,A -85,B 0,C 180,E1 -6344.983,E2 -6344.983} C_VEL
LIN {X 0,Y 488.763,Z 422.598,A -85,B 0,C 180,E1 -6345.668,E2 -6345.668} C_VEL
LIN {X 0,Y 488.688,Z 422.609,A -85,B 0,C 180,E1 -6345.9,E2 -6345.9} C_VEL
LIN {X 0,Y 488.669,Z 422.615,A -85,B 0,C 180,E1 -6348.58,E2 -6348.58} C_VEL
LIN {X 0,Y 488.691,Z 422.608,A -85,B 0,C 180,E1 -6350.949,E2 -6350.949} C_VEL
LIN {X 0,Y 488.655,Z 422.613,A -85,B 0,C 180,E1 -6353.866,E2 -6353.866} C_VEL
LIN {X 0,Y 488.74,Z 422.603,A -85,B 0,C 180,E1 -6356.877,E2 -6356.877} C_VEL
LIN {X 0,Y 488.721,Z 422.604,A -85,B 0,C 180,E1 -6359.78,E2 -6359.78} C_VEL
LIN {X 0,Y 488.702,Z 422.606,A -85,B 0,C 180,E1 -6363.077,E2 -6363.077} C_VEL
LIN {X 0,Y 488.672,Z 422.615,A -85,B 0,C 180,E1 -6366.253,E2 -6366.253} C_VEL
LIN {X 0,Y 488.749,Z 422.6,A -85,B 0,C 180,E1 -6369.175,E2 -6369.175} C_VEL
LIN {X 0,Y 488.749,Z 422.599,A -85,B 0,C 180,E1 -6371.632,E2 -6371.632} C_VEL
LIN {X 0,Y 488.757,Z 422.6,A -85,B 0,C 180,E1 -6374.999,E2 -6374.999} C_VEL
LIN {X 0,Y 488.807,Z 422.6,A -85,B 0,C 180,E1 -6378.387,E2 -6378.387} C_VEL
LIN {X 0,Y 488.781,Z 422.596,A -85,B 0,C 180,E1 -6381.733,E2 -6381.733} C_VEL
LIN {X 0,Y 488.831,Z 422.594,A -85,B 0,C 180,E1 -6384.224,E2 -6384.224} C_VEL
LIN {X 0,Y 488.955,Z 422.573,A -85,B 0,C 180,E1 -6387.528,E2 -6387.528} C_VEL
LIN {X 0,Y 488.915,Z 422.583,A -85,B 0,C 180,E1 -6390.823,E2 -6390.823} C_VEL
LIN {X 0,Y 488.953,Z 422.583,A -85,B 0,C 180,E1 -6392.471,E2 -6392.471} C_VEL
LIN {X 0,Y 488.853,Z 422.587,A -85,B 0,C 180,E1 -6395.775,E2 -6395.775} C_VEL
LIN {X 0,Y 488.785,Z 422.6,A -85,B 0,C 180,E1 -6398.267,E2 -6398.267} C_VEL
LIN {X 0,Y 488.806,Z 422.592,A -85,B 0,C 180,E1 -6401.612,E2 -6401.612} C_VEL
LIN {X 0,Y 488.765,Z 422.599,A -85,B 0,C 180,E1 -6405,E2 -6405} C_VEL
LIN {X 0,Y 488.748,Z 422.607,A -85,B 0,C 180,E1 -6408.442,E2 -6408.442} C_VEL
LIN {X 0,Y 488.708,Z 422.606,A -85,B 0,C 180,E1 -6411.07,E2 -6411.07} C_VEL
LIN {X 0,Y 488.676,Z 422.609,A -85,B 0,C 180,E1 -6413.746,E2 -6413.746} C_VEL
LIN {X 0,Y 488.717,Z 422.611,A -85,B 0,C 180,E1 -6416.474,E2 -6416.474} C_VEL
LIN {X 0,Y 488.71,Z 422.605,A -85,B 0,C 180,E1 -6419.271,E2 -6419.271} C_VEL
LIN {X 0,Y 488.703,Z 422.608,A -85,B 0,C 180,E1 -6422.147,E2 -6422.147} C_VEL
LIN {X 0,Y 488.716,Z 422.605,A -85,B 0,C 180,E1 -6425.115,E2 -6425.115} C_VEL
LIN {X 0,Y 488.675,Z 422.612,A -85,B 0,C 180,E1 -6428.2,E2 -6428.2} C_VEL
LIN {X 0,Y 488.718,Z 422.609,A -85,B 0,C 180,E1 -6430.344,E2 -6430.344} C_VEL
LIN {X 0,Y 488.676,Z 422.608,A -85,B 0,C 180,E1 -6433.655,E2 -6433.655} C_VEL
LIN {X 0,Y 488.678,Z 422.613,A -85,B 0,C 180,E1 -6436.344,E2 -6436.344} C_VEL
LIN {X 0,Y 488.717,Z 422.603,A -85,B 0,C 180,E1 -6439.675,E2 -6439.675} C_VEL
LIN {X 0,Y 488.67,Z 422.614,A -85,B 0,C 180,E1 -6442.84,E2 -6442.84} C_VEL
LIN {X 0,Y 488.729,Z 422.602,A -85,B 0,C 180,E1 -6445.887,E2 -6445.887} C_VEL
LIN {X 0,Y 488.692,Z 422.612,A -85,B 0,C 180,E1 -6448.82,E2 -6448.82} C_VEL
LIN {X 0,Y 488.741,Z 422.6,A -85,B 0,C 180,E1 -6451.671,E2 -6451.671} C_VEL
LIN {X 0,Y 488.715,Z 422.61,A -85,B 0,C 180,E1 -6454.442,E2 -6454.442} C_VEL
LIN {X 0,Y 488.721,Z 422.604,A -85,B 0,C 180,E1 -6457.153,E2 -6457.153} C_VEL
LIN {X 0,Y 488.724,Z 422.602,A -85,B 0,C 180,E1 -6459.81,E2 -6459.81} C_VEL
LIN {X 0,Y 488.714,Z 422.609,A -85,B 0,C 180,E1 -6462.423,E2 -6462.423} C_VEL
LIN {X 0,Y 488.761,Z 422.601,A -85,B 0,C 180,E1 -6465,E2 -6465} C_VEL
LIN {X 0,Y 488.805,Z 422.597,A -85,B 0,C 180,E1 -6468.388,E2 -6468.388} C_VEL
LIN {X 0,Y 488.816,Z 422.591,A -85,B 0,C 180,E1 -6471.734,E2 -6471.734} C_VEL
LIN {X 0,Y 488.806,Z 422.595,A -85,B 0,C 180,E1 -6475.051,E2 -6475.051} C_VEL
LIN {X 0,Y 488.96,Z 422.573,A -85,B 0,C 180,E1 -6477.529,E2 -6477.529} C_VEL
LIN {X 0,Y 488.934,Z 422.582,A -85,B 0,C 180,E1 -6480.824,E2 -6480.824} C_VEL
LIN {X 0,Y 488.961,Z 422.579,A -85,B 0,C 180,E1 -6482.471,E2 -6482.471} C_VEL
LIN {X 0,Y 488.853,Z 422.586,A -85,B 0,C 180,E1 -6485.776,E2 -6485.776} C_VEL
LIN {X 0,Y 488.816,Z 422.594,A -85,B 0,C 180,E1 -6488.266,E2 -6488.266} C_VEL
LIN {X 0,Y 488.806,Z 422.592,A -85,B 0,C 180,E1 -6491.613,E2 -6491.613} C_VEL
LIN {X 0,Y 488.765,Z 422.601,A -85,B 0,C 180,E1 -6495,E2 -6495} C_VEL
LIN {X 0,Y 488.747,Z 422.605,A -85,B 0,C 180,E1 -6498.443,E2 -6498.443} C_VEL
LIN {X 0,Y 488.707,Z 422.608,A -85,B 0,C 180,E1 -6501.071,E2 -6501.071} C_VEL
LIN {X 0,Y 488.687,Z 422.607,A -85,B 0,C 180,E1 -6503.746,E2 -6503.746} C_VEL
LIN {X 0,Y 488.737,Z 422.606,A -85,B 0,C 180,E1 -6506.473,E2 -6506.473} C_VEL
LIN {X 0,Y 488.722,Z 422.604,A -85,B 0,C 180,E1 -6509.271,E2 -6509.271} C_VEL
LIN {X 0,Y 488.703,Z 422.607,A -85,B 0,C 180,E1 -6512.147,E2 -6512.147} C_VEL
LIN {X 0,Y 488.717,Z 422.606,A -85,B 0,C 180,E1 -6515.115,E2 -6515.115} C_VEL
LIN {X 0,Y 488.68,Z 422.61,A -85,B 0,C 180,E1 -6518.2,E2 -6518.2} C_VEL
LIN {X 0,Y 488.718,Z 422.606,A -85,B 0,C 180,E1 -6520.345,E2 -6520.345} C_VEL
LIN {X 0,Y 488.687,Z 422.607,A -85,B 0,C 180,E1 -6523.655,E2 -6523.655} C_VEL
LIN {X 0,Y 488.688,Z 422.61,A -85,B 0,C 180,E1 -6526.346,E2 -6526.346} C_VEL
LIN {X 0,Y 488.734,Z 422.601,A -85,B 0,C 180,E1 -6529.677,E2 -6529.677} C_VEL
LIN {X 0,Y 488.671,Z 422.616,A -85,B 0,C 180,E1 -6532.841,E2 -6532.841} C_VEL
LIN {X 0,Y 488.731,Z 422.601,A -85,B 0,C 180,E1 -6535.887,E2 -6535.887} C_VEL
LIN {X 0,Y 488.693,Z 422.613,A -85,B 0,C 180,E1 -6538.821,E2 -6538.821} C_VEL
LIN {X 0,Y 488.747,Z 422.606,A -85,B 0,C 180,E1 -6542.139,E2 -6542.139} C_VEL
LIN {X 0,Y 488.77,Z 422.619,A -85,B 0,C 180,E1 -6542.605,E2 -6542.605} C_VEL
LIN {X 0,Y 491.227,Z 434.519,A -85,B 0,C 180,E1 -6544.583,E2 -6544.583} C_VEL
LIN {X 0,Y 491.238,Z 441.982,A -85,B 0,C 180,E1 -6545.735,E2 -6545.735} C_VEL
LIN {X 0,Y 490.349,Z 463.697,A -85,B 0,C 180,E1 -6549.003,E2 -6549.003} C_VEL
LIN {X 0,Y 489.722,Z 484.063,A -85,B 0,C 180,E1 -6552.029,E2 -6552.029} C_VEL
LIN {X 0,Y 489.339,Z 495.819,A -85,B 0,C 180,E1 -6553.736,E2 -6553.736} C_VEL
LIN {X 0,Y 491.577,Z 512.443,A -85,B 0,C 180,E1 -6554.075,E2 -6554.075} C_VEL
LIN {X 0,Y 490.844,Z 605.119,A -85,B 0,C 180,E1 -6555.516,E2 -6555.516} C_VEL
LIN {X 0,Y 490.619,Z 617.399,A -85,B 0,C 180,E1 -6555.853,E2 -6555.853} C_VEL
LIN {X 0,Y 490.23,Z 630.25,A -85,B 0,C 180,E1 -6556.37,E2 -6556.37} C_VEL
LIN {X 0,Y 489.839,Z 642.531,A -85,B 0,C 180,E1 -6557.046,E2 -6557.046} C_VEL
LIN {X 0,Y 489.453,Z 654.175,A -85,B 0,C 180,E1 -6557.878,E2 -6557.878} C_VEL
LIN {X 0,Y 489.073,Z 664.68,A -85,B 0,C 180,E1 -6558.814,E2 -6558.814} C_VEL
LIN {X 0,Y 488.727,Z 674.131,A -85,B 0,C 180,E1 -6559.854,E2 -6559.854} C_VEL
LIN {X 0,Y 488.399,Z 683.273,A -85,B 0,C 180,E1 -6561.101,E2 -6561.101} C_VEL
LIN {X 0,Y 488.215,Z 690.645,A -85,B 0,C 180,E1 -6562.348,E2 -6562.348} C_VEL
LIN {X 0,Y 488.076,Z 696.109,A -85,B 0,C 180,E1 -6563.495,E2 -6563.495} C_VEL
LIN {X 0,Y 488.055,Z 700.46,A -85,B 0,C 180,E1 -6564.63,E2 -6564.63} C_VEL
LIN {X 0,Y 487.996,Z 704.149,A -85,B 0,C 180,E1 -6565.871,E2 -6565.871} C_VEL
LIN {X 0,Y 487.974,Z 706.051,A -85,B 0,C 180,E1 -6566.698,E2 -6566.698} C_VEL
LIN {X 0,Y 487.989,Z 707.479,A -85,B 0,C 180,E1 -6567.524,E2 -6567.524} C_VEL
LIN {X 0,Y 487.85,Z 709.087,A -85,B 0,C 180,E1 -6569.175,E2 -6569.175} C_VEL
LIN {X 0,Y 487.85,Z 709.295,A -85,B 0,C 180,E1 -6570,E2 -6570} C_VEL
LIN {X 0,Y 487.852,Z 709.059,A -85,B 0,C 180,E1 -6570.826,E2 -6570.826} C_VEL
LIN {X 0,Y 487.991,Z 707.385,A -85,B 0,C 180,E1 -6572.477,E2 -6572.477} C_VEL
LIN {X 0,Y 487.986,Z 705.925,A -85,B 0,C 180,E1 -6573.303,E2 -6573.303} C_VEL
LIN {X 0,Y 487.955,Z 702.872,A -85,B 0,C 180,E1 -6574.544,E2 -6574.544} C_VEL
LIN {X 0,Y 488.078,Z 698.757,A -85,B 0,C 180,E1 -6575.785,E2 -6575.785} C_VEL
LIN {X 0,Y 488.183,Z 692.417,A -85,B 0,C 180,E1 -6577.237,E2 -6577.237} C_VEL
LIN {X 0,Y 488.341,Z 685.497,A -85,B 0,C 180,E1 -6578.483,E2 -6578.483} C_VEL
LIN {X 0,Y 488.565,Z 676.906,A -85,B 0,C 180,E1 -6579.731,E2 -6579.731} C_VEL
LIN {X 0,Y 488.898,Z 667.057,A -85,B 0,C 180,E1 -6580.876,E2 -6580.876} C_VEL
LIN {X 0,Y 489.257,Z 657.256,A -85,B 0,C 180,E1 -6581.804,E2 -6581.804} C_VEL
LIN {X 0,Y 489.586,Z 646.636,A -85,B 0,C 180,E1 -6582.624,E2 -6582.624} C_VEL
LIN {X 0,Y 489.986,Z 634.26,A -85,B 0,C 180,E1 -6583.373,E2 -6583.373} C_VEL
LIN {X 0,Y 490.374,Z 621.73,A -85,B 0,C 180,E1 -6583.943,E2 -6583.943} C_VEL
LIN {X 0,Y 490.69,Z 608.87,A -85,B 0,C 180,E1 -6584.357,E2 -6584.357} C_VEL
LIN {X 0,Y 490.957,Z 593.777,A -85,B 0,C 180,E1 -6584.64,E2 -6584.64} C_VEL
LIN {X 0,Y 491.483,Z 511.943,A -85,B 0,C 180,E1 -6585.912,E2 -6585.912} C_VEL
LIN {X 0,Y 489.258,Z 494.147,A -85,B 0,C 180,E1 -6586.29,E2 -6586.29} C_VEL
LIN {X 0,Y 489.86,Z 472.308,A -85,B 0,C 180,E1 -6589.486,E2 -6589.486} C_VEL
LIN {X 0,Y 490.432,Z 453.259,A -85,B 0,C 180,E1 -6592.319,E2 -6592.319} C_VEL
LIN {X 0,Y 491.09,Z 435.759,A -85,B 0,C 180,E1 -6594.972,E2 -6594.972} C_VEL
LIN {X 0,Y 490.244,Z 429.875,A -85,B 0,C 180,E1 -6595.928,E2 -6595.928} C_VEL
LIN {X 0,Y 488.772,Z 422.605,A -85,B 0,C 180,E1 -6597.195,E2 -6597.195} C_VEL
LIN {X 0,Y 488.714,Z 422.61,A -85,B 0,C 180,E1 -6600.363,E2 -6600.363} C_VEL
LIN {X 0,Y 488.739,Z 422.609,A -85,B 0,C 180,E1 -6603.484,E2 -6603.484} C_VEL
LIN {X 0,Y 488.686,Z 422.613,A -85,B 0,C 180,E1 -6606.355,E2 -6606.355} C_VEL
LIN {X 0,Y 488.705,Z 422.611,A -85,B 0,C 180,E1 -6609.254,E2 -6609.254} C_VEL
LIN {X 0,Y 488.71,Z 422.607,A -85,B 0,C 180,E1 -6611.6,E2 -6611.6} C_VEL
LIN {X 0,Y 488.705,Z 422.613,A -85,B 0,C 180,E1 -6614.803,E2 -6614.803} C_VEL
LIN {X 0,Y 488.692,Z 422.608,A -85,B 0,C 180,E1 -6617.474,E2 -6617.474} C_VEL
LIN {X 0,Y 488.704,Z 422.611,A -85,B 0,C 180,E1 -6620.746,E2 -6620.746} C_VEL
LIN {X 0,Y 488.673,Z 422.61,A -85,B 0,C 180,E1 -6623.867,E2 -6623.867} C_VEL
LIN {X 0,Y 488.742,Z 422.603,A -85,B 0,C 180,E1 -6626.877,E2 -6626.877} C_VEL
LIN {X 0,Y 488.722,Z 422.604,A -85,B 0,C 180,E1 -6629.78,E2 -6629.78} C_VEL
LIN {X 0,Y 488.701,Z 422.607,A -85,B 0,C 180,E1 -6633.079,E2 -6633.079} C_VEL
LIN {X 0,Y 488.673,Z 422.616,A -85,B 0,C 180,E1 -6636.253,E2 -6636.253} C_VEL
LIN {X 0,Y 488.677,Z 422.61,A -85,B 0,C 180,E1 -6639.199,E2 -6639.199} C_VEL
LIN {X 0,Y 488.661,Z 422.616,A -85,B 0,C 180,E1 -6642.421,E2 -6642.421} C_VEL
LIN {X 0,Y 488.718,Z 422.606,A -85,B 0,C 180,E1 -6644.998,E2 -6644.998} C_VEL
LIN {X 0,Y 488.776,Z 422.602,A -85,B 0,C 180,E1 -6648.387,E2 -6648.387} C_VEL
LIN {X 0,Y 488.757,Z 422.607,A -85,B 0,C 180,E1 -6651.733,E2 -6651.733} C_VEL
LIN {X 0,Y 488.806,Z 422.6,A -85,B 0,C 180,E1 -6654.224,E2 -6654.224} C_VEL
LIN {X 0,Y 488.958,Z 422.742,A -85,B 0,C 180,E1 -6657.58,E2 -6657.58} C_VEL
LIN {X 0,Y 489.524,Z 427.671,A -85,B 0,C 180,E1 -6658.826,E2 -6658.826} C_VEL
LIN {X 0,Y 491.844,Z 438.088,A -85,B 0,C 180,E1 -6659.09,E2 -6659.09} C_VEL
LIN {X 0,Y 490.949,Z 533.704,A -85,B 0,C 180,E1 -6660.615,E2 -6660.615} C_VEL
LIN {X 0,Y 490.747,Z 547.038,A -85,B 0,C 180,E1 -6661,E2 -6661} C_VEL
LIN {X 0,Y 490.524,Z 559.659,A -85,B 0,C 180,E1 -6661.539,E2 -6661.539} C_VEL
LIN {X 0,Y 490.21,Z 572.016,A -85,B 0,C 180,E1 -6662.259,E2 -6662.259} C_VEL
LIN {X 0,Y 489.713,Z 583.132,A -85,B 0,C 180,E1 -6663.085,E2 -6663.085} C_VEL
LIN {X 0,Y 489.414,Z 592.078,A -85,B 0,C 180,E1 -6663.911,E2 -6663.911} C_VEL
LIN {X 0,Y 489.065,Z 601.283,A -85,B 0,C 180,E1 -6664.946,E2 -6664.946} C_VEL
LIN {X 0,Y 488.779,Z 610.186,A -85,B 0,C 180,E1 -6666.191,E2 -6666.191} C_VEL
LIN {X 0,Y 488.563,Z 617.365,A -85,B 0,C 180,E1 -6667.439,E2 -6667.439} C_VEL
LIN {X 0,Y 488.328,Z 623.115,A -85,B 0,C 180,E1 -6668.692,E2 -6668.692} C_VEL
LIN {X 0,Y 488.175,Z 627.619,A -85,B 0,C 180,E1 -6669.948,E2 -6669.948} C_VEL
LIN {X 0,Y 488.128,Z 629.983,A -85,B 0,C 180,E1 -6670.788,E2 -6670.788} C_VEL
LIN {X 0,Y 488.091,Z 632.115,A -85,B 0,C 180,E1 -6671.724,E2 -6671.724} C_VEL
LIN {X 0,Y 487.977,Z 633.419,A -85,B 0,C 180,E1 -6672.476,E2 -6672.476} C_VEL
LIN {X 0,Y 487.938,Z 634.448,A -85,B 0,C 180,E1 -6673.324,E2 -6673.324} C_VEL
LIN {X 0,Y 487.94,Z 635.072,A -85,B 0,C 180,E1 -6674.173,E2 -6674.173} C_VEL
LIN {X 0,Y 487.929,Z 635.271,A -85,B 0,C 180,E1 -6675.191,E2 -6675.191} C_VEL
LIN {X 0,Y 487.894,Z 634.388,A -85,B 0,C 180,E1 -6676.744,E2 -6676.744} C_VEL
LIN {X 0,Y 488.004,Z 632.449,A -85,B 0,C 180,E1 -6678.102,E2 -6678.102} C_VEL
LIN {X 0,Y 488.08,Z 629.688,A -85,B 0,C 180,E1 -6679.341,E2 -6679.341} C_VEL
LIN {X 0,Y 488.213,Z 625.64,A -85,B 0,C 180,E1 -6680.658,E2 -6680.658} C_VEL
LIN {X 0,Y 488.341,Z 620.338,A -85,B 0,C 180,E1 -6681.974,E2 -6681.974} C_VEL
LIN {X 0,Y 488.587,Z 613.699,A -85,B 0,C 180,E1 -6683.263,E2 -6683.263} C_VEL
LIN {X 0,Y 488.854,Z 606.343,A -85,B 0,C 180,E1 -6684.414,E2 -6684.414} C_VEL
LIN {X 0,Y 489.193,Z 597.593,A -85,B 0,C 180,E1 -6685.531,E2 -6685.531} C_VEL
LIN {X 0,Y 489.537,Z 587.992,A -85,B 0,C 180,E1 -6686.532,E2 -6686.532} C_VEL
LIN {X 0,Y 489.931,Z 577.133,A -85,B 0,C 180,E1 -6687.441,E2 -6687.441} C_VEL
LIN {X 0,Y 490.319,Z 565.171,A -85,B 0,C 180,E1 -6688.23,E2 -6688.23} C_VEL
LIN {X 0,Y 490.631,Z 552.816,A -85,B 0,C 180,E1 -6688.852,E2 -6688.852} C_VEL
LIN {X 0,Y 490.862,Z 540.125,A -85,B 0,C 180,E1 -6689.307,E2 -6689.307} C_VEL
LIN {X 0,Y 491.036,Z 526.3,A -85,B 0,C 180,E1 -6689.619,E2 -6689.619} C_VEL
LIN {X 0,Y 491.699,Z 437.132,A -85,B 0,C 180,E1 -6690.999,E2 -6690.999} C_VEL
LIN {X 0,Y 489.25,Z 425.884,A -85,B 0,C 180,E1 -6691.272,E2 -6691.272} C_VEL
LIN {X 0,Y 488.759,Z 422.607,A -85,B 0,C 180,E1 -6692.08,E2 -6692.08} C_VEL
LIN {X 0,Y 488.713,Z 422.605,A -85,B 0,C 180,E1 -6695.115,E2 -6695.115} C_VEL
LIN {X 0,Y 488.661,Z 422.616,A -85,B 0,C 180,E1 -6698.202,E2 -6698.202} C_VEL
LIN {X 0,Y 488.696,Z 422.614,A -85,B 0,C 180,E1 -6700.341,E2 -6700.341} C_VEL
LIN {X 0,Y 488.677,Z 422.609,A -85,B 0,C 180,E1 -6703.656,E2 -6703.656} C_VEL
LIN {X 0,Y 488.688,Z 422.609,A -85,B 0,C 180,E1 -6705.9,E2 -6705.9} C_VEL
LIN {X 0,Y 488.04,Z 422.695,A -85,B 0,C 180,E1 -6706.588,E2 -6706.588} C_VEL
LIN {X 0,Y 485.183,Z 423.048,A -85,B 0,C 180,E1 -6707.705,E2 -6707.705} C_VEL
LIN {X 0,Y 482.758,Z 423.351,A -85,B 0,C 180,E1 -6708.605,E2 -6708.605} C_VEL
LIN {X 0,Y 481.719,Z 423.475,A -85,B 0,C 180,E1 -6709.3,E2 -6709.3} C_VEL
LIN {X 0,Y 481.638,Z 423.485,A -85,B 0,C 180,E1 -6709.536,E2 -6709.536} C_VEL
LIN {X 0,Y 481.607,Z 423.494,A -85,B 0,C 180,E1 -6712.2,E2 -6712.2} C_VEL
LIN {X 0,Y 481.685,Z 423.479,A -85,B 0,C 180,E1 -6715.317,E2 -6715.317} C_VEL
LIN {X 0,Y 481.647,Z 423.491,A -85,B 0,C 180,E1 -6718.311,E2 -6718.311} C_VEL
LIN {X 0,Y 481.662,Z 423.482,A -85,B 0,C 180,E1 -6721.216,E2 -6721.216} C_VEL
LIN {X 0,Y 481.648,Z 423.487,A -85,B 0,C 180,E1 -6724.039,E2 -6724.039} C_VEL
LIN {X 0,Y 481.676,Z 423.484,A -85,B 0,C 180,E1 -6726.812,E2 -6726.812} C_VEL
LIN {X 0,Y 481.697,Z 423.478,A -85,B 0,C 180,E1 -6729.502,E2 -6729.502} C_VEL
LIN {X 0,Y 481.683,Z 423.484,A -85,B 0,C 180,E1 -6732.157,E2 -6732.157} C_VEL
LIN {X 0,Y 481.74,Z 423.476,A -85,B 0,C 180,E1 -6734.775,E2 -6734.775} C_VEL
LIN {X 0,Y 481.753,Z 423.476,A -85,B 0,C 180,E1 -6738.215,E2 -6738.215} C_VEL
LIN {X 0,Y 481.737,Z 423.473,A -85,B 0,C 180,E1 -6741.611,E2 -6741.611} C_VEL
LIN {X 0,Y 481.79,Z 423.47,A -85,B 0,C 180,E1 -6744.139,E2 -6744.139} C_VEL
LIN {X 0,Y 481.921,Z 423.45,A -85,B 0,C 180,E1 -6747.492,E2 -6747.492} C_VEL
LIN {X 0,Y 481.94,Z 423.45,A -85,B 0,C 180,E1 -6750,E2 -6750} C_VEL
LIN {X 0,Y 481.919,Z 423.459,A -85,B 0,C 180,E1 -6752.507,E2 -6752.507} C_VEL
LIN {X 0,Y 481.814,Z 423.464,A -85,B 0,C 180,E1 -6755.86,E2 -6755.86} C_VEL
LIN {X 0,Y 481.74,Z 423.479,A -85,B 0,C 180,E1 -6758.388,E2 -6758.388} C_VEL
LIN {X 0,Y 481.752,Z 423.471,A -85,B 0,C 180,E1 -6761.785,E2 -6761.785} C_VEL
LIN {X 0,Y 481.745,Z 423.472,A -85,B 0,C 180,E1 -6765.224,E2 -6765.224} C_VEL
LIN {X 0,Y 481.709,Z 423.482,A -85,B 0,C 180,E1 -6768.722,E2 -6768.722} C_VEL
LIN {X 0,Y 481.646,Z 423.484,A -85,B 0,C 180,E1 -6771.394,E2 -6771.394} C_VEL
LIN {X 0,Y 481.657,Z 423.486,A -85,B 0,C 180,E1 -6774.114,E2 -6774.114} C_VEL
LIN {X 0,Y 481.694,Z 423.479,A -85,B 0,C 180,E1 -6777.127,E2 -6777.127} C_VEL
LIN {X 0,Y 481.673,Z 423.481,A -85,B 0,C 180,E1 -6779.741,E2 -6779.741} C_VEL
LIN {X 0,Y 481.672,Z 423.488,A -85,B 0,C 180,E1 -6782.674,E2 -6782.674} C_VEL
LIN {X 0,Y 481.634,Z 423.486,A -85,B 0,C 180,E1 -6785.71,E2 -6785.71} C_VEL
LIN {X 0,Y 481.667,Z 423.486,A -85,B 0,C 180,E1 -6788.859,E2 -6788.859} C_VEL
LIN {X 0,Y 481.646,Z 423.485,A -85,B 0,C 180,E1 -6791.912,E2 -6791.912} C_VEL
LIN {X 0,Y 481.653,Z 423.49,A -85,B 0,C 180,E1 -6794.458,E2 -6794.458} C_VEL
LIN {X 0,Y 481.642,Z 423.485,A -85,B 0,C 180,E1 -6797.839,E2 -6797.839} C_VEL
LIN {X 0,Y 481.66,Z 423.49,A -85,B 0,C 180,E1 -6800.654,E2 -6800.654} C_VEL
LIN {X 0,Y 481.621,Z 423.487,A -85,B 0,C 180,E1 -6803.377,E2 -6803.377} C_VEL
LIN {X 0,Y 481.709,Z 423.481,A -85,B 0,C 180,E1 -6806.33,E2 -6806.33} C_VEL
LIN {X 0,Y 481.65,Z 423.484,A -85,B 0,C 180,E1 -6809.417,E2 -6809.417} C_VEL
LIN {X 0,Y 481.691,Z 423.481,A -85,B 0,C 180,E1 -6812.167,E2 -6812.167} C_VEL
LIN {X 0,Y 481.688,Z 423.482,A -85,B 0,C 180,E1 -6814.968,E2 -6814.968} C_VEL
LIN {X 0,Y 481.648,Z 423.484,A -85,B 0,C 180,E1 -6817.705,E2 -6817.705} C_VEL
LIN {X 0,Y 481.704,Z 423.482,A -85,B 0,C 180,E1 -6820.393,E2 -6820.393} C_VEL
LIN {X 0,Y 481.678,Z 423.483,A -85,B 0,C 180,E1 -6823.033,E2 -6823.033} C_VEL
LIN {X 0,Y 481.687,Z 423.479,A -85,B 0,C 180,E1 -6825.639,E2 -6825.639} C_VEL
LIN {X 0,Y 481.751,Z 423.474,A -85,B 0,C 180,E1 -6828.215,E2 -6828.215} C_VEL
LIN {X 0,Y 481.761,Z 423.47,A -85,B 0,C 180,E1 -6831.612,E2 -6831.612} C_VEL
LIN {X 0,Y 481.776,Z 423.472,A -85,B 0,C 180,E1 -6834.979,E2 -6834.979} C_VEL
LIN {X 0,Y 481.927,Z 423.449,A -85,B 0,C 180,E1 -6837.493,E2 -6837.493} C_VEL
LIN {X 0,Y 481.885,Z 423.46,A -85,B 0,C 180,E1 -6840.836,E2 -6840.836} C_VEL
LIN {X 0,Y 481.927,Z 423.456,A -85,B 0,C 180,E1 -6842.508,E2 -6842.508} C_VEL
LIN {X 0,Y 481.815,Z 423.463,A -85,B 0,C 180,E1 -6845.861,E2 -6845.861} C_VEL
LIN {X 0,Y 481.761,Z 423.474,A -85,B 0,C 180,E1 -6848.388,E2 -6848.388} C_VEL
LIN {X 0,Y 481.751,Z 423.471,A -85,B 0,C 180,E1 -6851.785,E2 -6851.785} C_VEL
LIN {X 0,Y 481.744,Z 423.474,A -85,B 0,C 180,E1 -6855.224,E2 -6855.224} C_VEL
LIN {X 0,Y 481.708,Z 423.485,A -85,B 0,C 180,E1 -6858.722,E2 -6858.722} C_VEL
LIN {X 0,Y 481.645,Z 423.485,A -85,B 0,C 180,E1 -6861.395,E2 -6861.395} C_VEL
LIN {X 0,Y 481.671,Z 423.482,A -85,B 0,C 180,E1 -6864.114,E2 -6864.114} C_VEL
LIN {X 0,Y 481.713,Z 423.479,A -85,B 0,C 180,E1 -6867.132,E2 -6867.132} C_VEL
LIN {X 0,Y 481.678,Z 423.48,A -85,B 0,C 180,E1 -6869.741,E2 -6869.741} C_VEL
LIN {X 0,Y 481.672,Z 423.489,A -85,B 0,C 180,E1 -6872.674,E2 -6872.674} C_VEL
LIN {X 0,Y 481.637,Z 423.485,A -85,B 0,C 180,E1 -6875.71,E2 -6875.71} C_VEL
LIN {X 0,Y 481.671,Z 423.488,A -85,B 0,C 180,E1 -6878.859,E2 -6878.859} C_VEL
LIN {X 0,Y 481.652,Z 423.483,A -85,B 0,C 180,E1 -6881.913,E2 -6881.913} C_VEL
LIN {X 0,Y 481.66,Z 423.487,A -85,B 0,C 180,E1 -6884.458,E2 -6884.458} C_VEL
LIN {X 0,Y 481.648,Z 423.484,A -85,B 0,C 180,E1 -6887.84,E2 -6887.84} C_VEL
LIN {X 0,Y 481.681,Z 423.487,A -85,B 0,C 180,E1 -6890.651,E2 -6890.651} C_VEL
LIN {X 0,Y 481.622,Z 423.488,A -85,B 0,C 180,E1 -6893.377,E2 -6893.377} C_VEL
LIN {X 0,Y 481.711,Z 423.479,A -85,B 0,C 180,E1 -6896.33,E2 -6896.33} C_VEL
LIN {X 0,Y 481.652,Z 423.486,A -85,B 0,C 180,E1 -6899.418,E2 -6899.418} C_VEL
LIN {X 0,Y 481.732,Z 423.494,A -85,B 0,C 180,E1 -6902.391,E2 -6902.391} C_VEL
LIN {X 0,Y 484.41,Z 436.983,A -85,B 0,C 180,E1 -6904.66,E2 -6904.66} C_VEL
LIN {X 0,Y 484.002,Z 448.997,A -85,B 0,C 180,E1 -6906.515,E2 -6906.515} C_VEL
LIN {X 0,Y 483.265,Z 467.603,A -85,B 0,C 180,E1 -6909.35,E2 -6909.35} C_VEL
LIN {X 0,Y 482.621,Z 486.497,A -85,B 0,C 180,E1 -6912.194,E2 -6912.194} C_VEL
LIN {X 0,Y 482.351,Z 495.387,A -85,B 0,C 180,E1 -6913.498,E2 -6913.498} C_VEL
LIN {X 0,Y 484.753,Z 514.193,A -85,B 0,C 180,E1 -6913.882,E2 -6913.882} C_VEL
LIN {X 0,Y 483.948,Z 605.166,A -85,B 0,C 180,E1 -6915.331,E2 -6915.331} C_VEL
LIN {X 0,Y 483.68,Z 618.014,A -85,B 0,C 180,E1 -6915.699,E2 -6915.699} C_VEL
LIN {X 0,Y 483.261,Z 630.573,A -85,B 0,C 180,E1 -6916.224,E2 -6916.224} C_VEL
LIN {X 0,Y 482.884,Z 641.814,A -85,B 0,C 180,E1 -6916.856,E2 -6916.856} C_VEL
LIN {X 0,Y 482.449,Z 653.592,A -85,B 0,C 180,E1 -6917.707,E2 -6917.707} C_VEL
LIN {X 0,Y 482.059,Z 664.032,A -85,B 0,C 180,E1 -6918.649,E2 -6918.649} C_VEL
LIN {X 0,Y 481.683,Z 673.518,A -85,B 0,C 180,E1 -6919.704,E2 -6919.704} C_VEL
LIN {X 0,Y 481.34,Z 682.682,A -85,B 0,C 180,E1 -6920.97,E2 -6920.97} C_VEL
LIN {X 0,Y 481.142,Z 690.071,A -85,B 0,C 180,E1 -6922.235,E2 -6922.235} C_VEL
LIN {X 0,Y 480.975,Z 696.088,A -85,B 0,C 180,E1 -6923.524,E2 -6923.524} C_VEL
LIN {X 0,Y 480.906,Z 701.26,A -85,B 0,C 180,E1 -6924.97,E2 -6924.97} C_VEL
LIN {X 0,Y 480.894,Z 703.608,A -85,B 0,C 180,E1 -6925.81,E2 -6925.81} C_VEL
LIN {X 0,Y 480.902,Z 705.515,A -85,B 0,C 180,E1 -6926.649,E2 -6926.649} C_VEL
LIN {X 0,Y 480.926,Z 706.948,A -85,B 0,C 180,E1 -6927.488,E2 -6927.488} C_VEL
LIN {X 0,Y 480.775,Z 708.554,A -85,B 0,C 180,E1 -6929.163,E2 -6929.163} C_VEL
LIN {X 0,Y 480.772,Z 708.76,A -85,B 0,C 180,E1 -6930,E2 -6930} C_VEL
LIN {X 0,Y 480.776,Z 708.521,A -85,B 0,C 180,E1 -6930.838,E2 -6930.838} C_VEL
LIN {X 0,Y 480.928,Z 706.833,A -85,B 0,C 180,E1 -6932.513,E2 -6932.513} C_VEL
LIN {X 0,Y 480.914,Z 705.364,A -85,B 0,C 180,E1 -6933.351,E2 -6933.351} C_VEL
LIN {X 0,Y 480.868,Z 702.294,A -85,B 0,C 180,E1 -6934.611,E2 -6934.611} C_VEL
LIN {X 0,Y 480.973,Z 698.156,A -85,B 0,C 180,E1 -6935.871,E2 -6935.871} C_VEL
LIN {X 0,Y 481.108,Z 691.785,A -85,B 0,C 180,E1 -6937.344,E2 -6937.344} C_VEL
LIN {X 0,Y 481.278,Z 684.837,A -85,B 0,C 180,E1 -6938.609,E2 -6938.609} C_VEL
LIN {X 0,Y 481.502,Z 676.21,A -85,B 0,C 180,E1 -6939.876,E2 -6939.876} C_VEL
LIN {X 0,Y 481.891,Z 666.325,A -85,B 0,C 180,E1 -6941.036,E2 -6941.036} C_VEL
LIN {X 0,Y 482.285,Z 655.75,A -85,B 0,C 180,E1 -6942.042,E2 -6942.042} C_VEL
LIN {X 0,Y 482.607,Z 645.513,A -85,B 0,C 180,E1 -6942.832,E2 -6942.832} C_VEL
LIN {X 0,Y 483.033,Z 633.347,A -85,B 0,C 180,E1 -6943.569,E2 -6943.569} C_VEL
LIN {X 0,Y 483.457,Z 620.728,A -85,B 0,C 180,E1 -6944.147,E2 -6944.147} C_VEL
LIN {X 0,Y 483.821,Z 607.663,A -85,B 0,C 180,E1 -6944.566,E2 -6944.566} C_VEL
LIN {X 0,Y 484.062,Z 592.353,A -85,B 0,C 180,E1 -6944.854,E2 -6944.854} C_VEL
LIN {X 0,Y 484.619,Z 512.264,A -85,B 0,C 180,E1 -6946.13,E2 -6946.13} C_VEL
LIN {X 0,Y 482.261,Z 493.521,A -85,B 0,C 180,E1 -6946.537,E2 -6946.537} C_VEL
LIN {X 0,Y 482.913,Z 471.776,A -85,B 0,C 180,E1 -6949.778,E2 -6949.778} C_VEL
LIN {X 0,Y 483.487,Z 454.242,A -85,B 0,C 180,E1 -6952.431,E2 -6952.431} C_VEL
LIN {X 0,Y 484.176,Z 436.872,A -85,B 0,C 180,E1 -6955.113,E2 -6955.113} C_VEL
LIN {X 0,Y 482.969,Z 429.504,A -85,B 0,C 180,E1 -6956.349,E2 -6956.349} C_VEL
LIN {X 0,Y 481.727,Z 423.482,A -85,B 0,C 180,E1 -6957.398,E2 -6957.398} C_VEL
LIN {X 0,Y 481.655,Z 423.491,A -85,B 0,C 180,E1 -6960.583,E2 -6960.583} C_VEL
LIN {X 0,Y 481.701,Z 423.485,A -85,B 0,C 180,E1 -6963.733,E2 -6963.733} C_VEL
LIN {X 0,Y 481.629,Z 423.495,A -85,B 0,C 180,E1 -6966.747,E2 -6966.747} C_VEL
LIN {X 0,Y 481.681,Z 423.483,A -85,B 0,C 180,E1 -6969.941,E2 -6969.941} C_VEL
LIN {X 0,Y 481.642,Z 423.488,A -85,B 0,C 180,E1 -6973.3,E2 -6973.3} C_VEL
LIN {X 0,Y 481.656,Z 423.484,A -85,B 0,C 180,E1 -6975.642,E2 -6975.642} C_VEL
LIN {X 0,Y 481.653,Z 423.488,A -85,B 0,C 180,E1 -6978.958,E2 -6978.958} C_VEL
LIN {X 0,Y 481.654,Z 423.486,A -85,B 0,C 180,E1 -6981.994,E2 -6981.994} C_VEL
LIN {X 0,Y 481.691,Z 423.479,A -85,B 0,C 180,E1 -6985.318,E2 -6985.318} C_VEL
LIN {X 0,Y 481.648,Z 423.49,A -85,B 0,C 180,E1 -6988.312,E2 -6988.312} C_VEL
LIN {X 0,Y 481.664,Z 423.483,A -85,B 0,C 180,E1 -6991.216,E2 -6991.216} C_VEL
LIN {X 0,Y 481.646,Z 423.49,A -85,B 0,C 180,E1 -6994.04,E2 -6994.04} C_VEL
LIN {X 0,Y 481.678,Z 423.484,A -85,B 0,C 180,E1 -6996.812,E2 -6996.812} C_VEL
LIN {X 0,Y 481.622,Z 423.49,A -85,B 0,C 180,E1 -6999.499,E2 -6999.499} C_VEL
LIN {X 0,Y 481.646,Z 423.492,A -85,B 0,C 180,E1 -7002.156,E2 -7002.156} C_VEL
LIN {X 0,Y 481.694,Z 423.482,A -85,B 0,C 180,E1 -7004.774,E2 -7004.774} C_VEL
LIN {X 0,Y 481.728,Z 423.482,A -85,B 0,C 180,E1 -7008.214,E2 -7008.214} C_VEL
LIN {X 0,Y 481.715,Z 423.483,A -85,B 0,C 180,E1 -7011.611,E2 -7011.611} C_VEL
LIN {X 0,Y 481.767,Z 423.477,A -85,B 0,C 180,E1 -7014.139,E2 -7014.139} C_VEL
LIN {X 0,Y 481.852,Z 423.516,A -85,B 0,C 180,E1 -7017.335,E2 -7017.335} C_VEL
LIN {X 0,Y 482.549,Z 428.309,A -85,B 0,C 180,E1 -7018.569,E2 -7018.569} C_VEL
LIN {X 0,Y 485.034,Z 438.341,A -85,B 0,C 180,E1 -7018.848,E2 -7018.848} C_VEL
LIN {X 0,Y 484.071,Z 534.167,A -85,B 0,C 180,E1 -7020.416,E2 -7020.416} C_VEL
LIN {X 0,Y 483.843,Z 548.264,A -85,B 0,C 180,E1 -7020.832,E2 -7020.832} C_VEL
LIN {X 0,Y 483.649,Z 560.158,A -85,B 0,C 180,E1 -7021.353,E2 -7021.353} C_VEL
LIN {X 0,Y 483.301,Z 572.542,A -85,B 0,C 180,E1 -7022.083,E2 -7022.083} C_VEL
LIN {X 0,Y 482.793,Z 583.667,A -85,B 0,C 180,E1 -7022.92,E2 -7022.92} C_VEL
LIN {X 0,Y 482.454,Z 592.634,A -85,B 0,C 180,E1 -7023.759,E2 -7023.759} C_VEL
LIN {X 0,Y 482.096,Z 601.845,A -85,B 0,C 180,E1 -7024.808,E2 -7024.808} C_VEL
LIN {X 0,Y 481.78,Z 610.757,A -85,B 0,C 180,E1 -7026.071,E2 -7026.071} C_VEL
LIN {X 0,Y 481.544,Z 617.857,A -85,B 0,C 180,E1 -7027.321,E2 -7027.321} C_VEL
LIN {X 0,Y 481.325,Z 622.801,A -85,B 0,C 180,E1 -7028.396,E2 -7028.396} C_VEL
LIN {X 0,Y 481.171,Z 627.503,A -85,B 0,C 180,E1 -7029.67,E2 -7029.67} C_VEL
LIN {X 0,Y 481.077,Z 631.081,A -85,B 0,C 180,E1 -7030.948,E2 -7030.948} C_VEL
LIN {X 0,Y 481.008,Z 632.901,A -85,B 0,C 180,E1 -7031.803,E2 -7031.803} C_VEL
LIN {X 0,Y 480.895,Z 634.257,A -85,B 0,C 180,E1 -7032.663,E2 -7032.663} C_VEL
LIN {X 0,Y 480.866,Z 635.198,A -85,B 0,C 180,E1 -7033.524,E2 -7033.524} C_VEL
LIN {X 0,Y 480.863,Z 635.729,A -85,B 0,C 180,E1 -7034.386,E2 -7034.386} C_VEL
LIN {X 0,Y 480.865,Z 635.787,A -85,B 0,C 180,E1 -7035.287,E2 -7035.287} C_VEL
LIN {X 0,Y 480.841,Z 635.448,A -85,B 0,C 180,E1 -7036.123,E2 -7036.123} C_VEL
LIN {X 0,Y 480.827,Z 634.689,A -85,B 0,C 180,E1 -7036.997,E2 -7036.997} C_VEL
LIN {X 0,Y 480.937,Z 632.835,A -85,B 0,C 180,E1 -7038.22,E2 -7038.22} C_VEL
LIN {X 0,Y 481.027,Z 629.593,A -85,B 0,C 180,E1 -7039.636,E2 -7039.636} C_VEL
LIN {X 0,Y 481.188,Z 624.971,A -85,B 0,C 180,E1 -7041.059,E2 -7041.059} C_VEL
LIN {X 0,Y 481.396,Z 618.693,A -85,B 0,C 180,E1 -7042.517,E2 -7042.517} C_VEL
LIN {X 0,Y 481.692,Z 611.154,A -85,B 0,C 180,E1 -7043.884,E2 -7043.884} C_VEL
LIN {X 0,Y 482.023,Z 603.365,A -85,B 0,C 180,E1 -7045.013,E2 -7045.013} C_VEL
LIN {X 0,Y 482.383,Z 593.753,A -85,B 0,C 180,E1 -7046.15,E2 -7046.15} C_VEL
LIN {X 0,Y 482.781,Z 583.189,A -85,B 0,C 180,E1 -7047.157,E2 -7047.157} C_VEL
LIN {X 0,Y 483.161,Z 572.4,A -85,B 0,C 180,E1 -7047.976,E2 -7047.976} C_VEL
LIN {X 0,Y 483.54,Z 560.963,A -85,B 0,C 180,E1 -7048.662,E2 -7048.662} C_VEL
LIN {X 0,Y 483.869,Z 548.892,A -85,B 0,C 180,E1 -7049.212,E2 -7049.212} C_VEL
LIN {X 0,Y 484.062,Z 536.44,A -85,B 0,C 180,E1 -7049.61,E2 -7049.61} C_VEL
LIN {X 0,Y 484.214,Z 519.216,A -85,B 0,C 180,E1 -7049.929,E2 -7049.929} C_VEL
LIN {X 0,Y 484.87,Z 437.942,A -85,B 0,C 180,E1 -7051.219,E2 -7051.219} C_VEL
LIN {X 0,Y 482.174,Z 426.306,A -85,B 0,C 180,E1 -7051.512,E2 -7051.512} C_VEL
LIN {X 0,Y 481.715,Z 423.484,A -85,B 0,C 180,E1 -7052.199,E2 -7052.199} C_VEL
LIN {X 0,Y 481.657,Z 423.484,A -85,B 0,C 180,E1 -7055.203,E2 -7055.203} C_VEL
LIN {X 0,Y 481.637,Z 423.488,A -85,B 0,C 180,E1 -7058.004,E2 -7058.004} C_VEL
LIN {X 0,Y 481.634,Z 423.487,A -85,B 0,C 180,E1 -7061.044,E2 -7061.044} C_VEL
LIN {X 0,Y 481.656,Z 423.491,A -85,B 0,C 180,E1 -7064.458,E2 -7064.458} C_VEL
LIN {X 0,Y 481.618,Z 423.49,A -85,B 0,C 180,E1 -7066.855,E2 -7066.855} C_VEL
LIN {X 0,Y 481.638,Z 423.485,A -85,B 0,C 180,E1 -7069.536,E2 -7069.536} C_VEL
LIN {X 0,Y 480.971,Z 423.575,A -85,B 0,C 180,E1 -7070.234,E2 -7070.234} C_VEL
LIN {X 0,Y 478.097,Z 423.93,A -85,B 0,C 180,E1 -7071.367,E2 -7071.367} C_VEL
LIN {X 0,Y 475.669,Z 424.235,A -85,B 0,C 180,E1 -7072.28,E2 -7072.28} C_VEL
LIN {X 0,Y 474.635,Z 424.359,A -85,B 0,C 180,E1 -7072.986,E2 -7072.986} C_VEL
LIN {X 0,Y 474.556,Z 424.367,A -85,B 0,C 180,E1 -7073.225,E2 -7073.225} C_VEL
LIN {X 0,Y 474.638,Z 424.36,A -85,B 0,C 180,E1 -7076.016,E2 -7076.016} C_VEL
LIN {X 0,Y 474.603,Z 424.362,A -85,B 0,C 180,E1 -7079.19,E2 -7079.19} C_VEL
LIN {X 0,Y 474.608,Z 424.361,A -85,B 0,C 180,E1 -7081.715,E2 -7081.715} C_VEL
LIN {X 0,Y 474.629,Z 424.365,A -85,B 0,C 180,E1 -7084.589,E2 -7084.589} C_VEL
LIN {X 0,Y 474.602,Z 424.362,A -85,B 0,C 180,E1 -7087.355,E2 -7087.355} C_VEL
LIN {X 0,Y 474.654,Z 424.359,A -85,B 0,C 180,E1 -7090.089,E2 -7090.089} C_VEL
LIN {X 0,Y 474.626,Z 424.363,A -85,B 0,C 180,E1 -7092.773,E2 -7092.773} C_VEL
LIN {X 0,Y 474.641,Z 424.357,A -85,B 0,C 180,E1 -7095.42,E2 -7095.42} C_VEL
LIN {X 0,Y 474.707,Z 424.351,A -85,B 0,C 180,E1 -7098.037,E2 -7098.037} C_VEL
LIN {X 0,Y 474.71,Z 424.348,A -85,B 0,C 180,E1 -7101.486,E2 -7101.486} C_VEL
LIN {X 0,Y 474.751,Z 424.346,A -85,B 0,C 180,E1 -7104.052,E2 -7104.052} C_VEL
LIN {X 0,Y 474.887,Z 424.326,A -85,B 0,C 180,E1 -7107.455,E2 -7107.455} C_VEL
LIN {X 0,Y 474.91,Z 424.325,A -85,B 0,C 180,E1 -7110,E2 -7110} C_VEL
LIN {X 0,Y 474.884,Z 424.334,A -85,B 0,C 180,E1 -7112.544,E2 -7112.544} C_VEL
LIN {X 0,Y 474.777,Z 424.341,A -85,B 0,C 180,E1 -7115.947,E2 -7115.947} C_VEL
LIN {X 0,Y 474.711,Z 424.357,A -85,B 0,C 180,E1 -7118.514,E2 -7118.514} C_VEL
LIN {X 0,Y 474.706,Z 424.35,A -85,B 0,C 180,E1 -7121.962,E2 -7121.962} C_VEL
LIN {X 0,Y 474.701,Z 424.349,A -85,B 0,C 180,E1 -7125.455,E2 -7125.455} C_VEL
LIN {X 0,Y 474.664,Z 424.356,A -85,B 0,C 180,E1 -7129.01,E2 -7129.01} C_VEL
LIN {X 0,Y 474.589,Z 424.363,A -85,B 0,C 180,E1 -7131.729,E2 -7131.729} C_VEL
LIN {X 0,Y 474.637,Z 424.365,A -85,B 0,C 180,E1 -7134.494,E2 -7134.494} C_VEL
LIN {X 0,Y 474.637,Z 424.357,A -85,B 0,C 180,E1 -7137.324,E2 -7137.324} C_VEL
LIN {X 0,Y 474.603,Z 424.366,A -85,B 0,C 180,E1 -7140.23,E2 -7140.23} C_VEL
LIN {X 0,Y 474.643,Z 424.357,A -85,B 0,C 180,E1 -7143.22,E2 -7143.22} C_VEL
LIN {X 0,Y 474.585,Z 424.369,A -85,B 0,C 180,E1 -7146.324,E2 -7146.324} C_VEL
LIN {X 0,Y 474.623,Z 424.359,A -85,B 0,C 180,E1 -7149.548,E2 -7149.548} C_VEL
LIN {X 0,Y 474.599,Z 424.366,A -85,B 0,C 180,E1 -7152.233,E2 -7152.233} C_VEL
LIN {X 0,Y 474.615,Z 424.36,A -85,B 0,C 180,E1 -7155.298,E2 -7155.298} C_VEL
LIN {X 0,Y 474.614,Z 424.364,A -85,B 0,C 180,E1 -7158.214,E2 -7158.214} C_VEL
LIN {X 0,Y 474.609,Z 424.361,A -85,B 0,C 180,E1 -7161.542,E2 -7161.542} C_VEL
LIN {X 0,Y 474.621,Z 424.366,A -85,B 0,C 180,E1 -7164.725,E2 -7164.725} C_VEL
LIN {X 0,Y 474.635,Z 424.358,A -85,B 0,C 180,E1 -7167.788,E2 -7167.788} C_VEL
LIN {X 0,Y 474.622,Z 424.364,A -85,B 0,C 180,E1 -7170.885,E2 -7170.885} C_VEL
LIN {X 0,Y 474.629,Z 424.358,A -85,B 0,C 180,E1 -7173.626,E2 -7173.626} C_VEL
LIN {X 0,Y 474.634,Z 424.366,A -85,B 0,C 180,E1 -7176.642,E2 -7176.642} C_VEL
LIN {X 0,Y 474.654,Z 424.357,A -85,B 0,C 180,E1 -7180.09,E2 -7180.09} C_VEL
LIN {X 0,Y 474.637,Z 424.363,A -85,B 0,C 180,E1 -7182.774,E2 -7182.774} C_VEL
LIN {X 0,Y 474.646,Z 424.356,A -85,B 0,C 180,E1 -7185.421,E2 -7185.421} C_VEL
LIN {X 0,Y 474.704,Z 424.35,A -85,B 0,C 180,E1 -7188.038,E2 -7188.038} C_VEL
LIN {X 0,Y 474.726,Z 424.346,A -85,B 0,C 180,E1 -7191.486,E2 -7191.486} C_VEL
LIN {X 0,Y 474.747,Z 424.348,A -85,B 0,C 180,E1 -7194.904,E2 -7194.904} C_VEL
LIN {X 0,Y 474.893,Z 424.326,A -85,B 0,C 180,E1 -7197.455,E2 -7197.455} C_VEL
LIN {X 0,Y 474.911,Z 424.324,A -85,B 0,C 180,E1 -7200,E2 -7200} C_VEL
LIN {X 0,Y 474.893,Z 424.332,A -85,B 0,C 180,E1 -7202.545,E2 -7202.545} C_VEL
LIN {X 0,Y 474.778,Z 424.34,A -85,B 0,C 180,E1 -7205.948,E2 -7205.948} C_VEL
LIN {X 0,Y 474.726,Z 424.352,A -85,B 0,C 180,E1 -7208.514,E2 -7208.514} C_VEL
LIN {X 0,Y 474.704,Z 424.349,A -85,B 0,C 180,E1 -7211.963,E2 -7211.963} C_VEL
LIN {X 0,Y 474.701,Z 424.35,A -85,B 0,C 180,E1 -7215.456,E2 -7215.456} C_VEL
LIN {X 0,Y 474.663,Z 424.358,A -85,B 0,C 180,E1 -7219.01,E2 -7219.01} C_VEL
LIN {X 0,Y 474.588,Z 424.363,A -85,B 0,C 180,E1 -7221.729,E2 -7221.729} C_VEL
LIN {X 0,Y 474.65,Z 424.361,A -85,B 0,C 180,E1 -7224.493,E2 -7224.493} C_VEL
LIN {X 0,Y 474.673,Z 424.354,A -85,B 0,C 180,E1 -7227.333,E2 -7227.333} C_VEL
LIN {X 0,Y 474.605,Z 424.364,A -85,B 0,C 180,E1 -7230.23,E2 -7230.23} C_VEL
LIN {X 0,Y 474.643,Z 424.359,A -85,B 0,C 180,E1 -7233.22,E2 -7233.22} C_VEL
LIN {X 0,Y 474.589,Z 424.366,A -85,B 0,C 180,E1 -7236.324,E2 -7236.324} C_VEL
LIN {X 0,Y 474.618,Z 424.359,A -85,B 0,C 180,E1 -7239.646,E2 -7239.646} C_VEL
LIN {X 0,Y 474.615,Z 424.366,A -85,B 0,C 180,E1 -7242.934,E2 -7242.934} C_VEL
LIN {X 0,Y 474.614,Z 424.36,A -85,B 0,C 180,E1 -7245.896,E2 -7245.896} C_VEL
LIN {X 0,Y 474.628,Z 424.363,A -85,B 0,C 180,E1 -7249.041,E2 -7249.041} C_VEL
LIN {X 0,Y 474.608,Z 424.361,A -85,B 0,C 180,E1 -7251.705,E2 -7251.705} C_VEL
LIN {X 0,Y 474.623,Z 424.367,A -85,B 0,C 180,E1 -7254.726,E2 -7254.726} C_VEL
LIN {X 0,Y 474.637,Z 424.357,A -85,B 0,C 180,E1 -7257.788,E2 -7257.788} C_VEL
LIN {X 0,Y 474.624,Z 424.366,A -85,B 0,C 180,E1 -7260.885,E2 -7260.885} C_VEL
LIN {X 0,Y 474.717,Z 424.53,A -85,B 0,C 180,E1 -7262.2,E2 -7262.2} C_VEL
LIN {X 0,Y 477.466,Z 438.228,A -85,B 0,C 180,E1 -7264.542,E2 -7264.542} C_VEL
LIN {X 0,Y 477.128,Z 449.041,A -85,B 0,C 180,E1 -7266.241,E2 -7266.241} C_VEL
LIN {X 0,Y 476.293,Z 468.583,A -85,B 0,C 180,E1 -7269.26,E2 -7269.26} C_VEL
LIN {X 0,Y 475.601,Z 487.471,A -85,B 0,C 180,E1 -7272.144,E2 -7272.144} C_VEL
LIN {X 0,Y 475.366,Z 494.725,A -85,B 0,C 180,E1 -7273.246,E2 -7273.246} C_VEL
LIN {X 0,Y 477.916,Z 513.771,A -85,B 0,C 180,E1 -7273.655,E2 -7273.655} C_VEL
LIN {X 0,Y 477.103,Z 603.964,A -85,B 0,C 180,E1 -7275.116,E2 -7275.116} C_VEL
LIN {X 0,Y 476.757,Z 616.258,A -85,B 0,C 180,E1 -7275.46,E2 -7275.46} C_VEL
LIN {X 0,Y 476.288,Z 629.692,A -85,B 0,C 180,E1 -7276.018,E2 -7276.018} C_VEL
LIN {X 0,Y 475.918,Z 641.043,A -85,B 0,C 180,E1 -7276.66,E2 -7276.66} C_VEL
LIN {X 0,Y 475.465,Z 652.188,A -85,B 0,C 180,E1 -7277.466,E2 -7277.466} C_VEL
LIN {X 0,Y 475.027,Z 663.36,A -85,B 0,C 180,E1 -7278.479,E2 -7278.479} C_VEL
LIN {X 0,Y 474.621,Z 672.891,A -85,B 0,C 180,E1 -7279.549,E2 -7279.549} C_VEL
LIN {X 0,Y 474.275,Z 682.083,A -85,B 0,C 180,E1 -7280.834,E2 -7280.834} C_VEL
LIN {X 0,Y 474.064,Z 689.493,A -85,B 0,C 180,E1 -7282.118,E2 -7282.118} C_VEL
LIN {X 0,Y 473.936,Z 694.503,A -85,B 0,C 180,E1 -7283.187,E2 -7283.187} C_VEL
LIN {X 0,Y 473.895,Z 699.363,A -85,B 0,C 180,E1 -7284.469,E2 -7284.469} C_VEL
LIN {X 0,Y 473.796,Z 703.066,A -85,B 0,C 180,E1 -7285.747,E2 -7285.747} C_VEL
LIN {X 0,Y 473.83,Z 704.98,A -85,B 0,C 180,E1 -7286.599,E2 -7286.599} C_VEL
LIN {X 0,Y 473.865,Z 706.416,A -85,B 0,C 180,E1 -7287.45,E2 -7287.45} C_VEL
LIN {X 0,Y 473.703,Z 708.021,A -85,B 0,C 180,E1 -7289.15,E2 -7289.15} C_VEL
LIN {X 0,Y 473.697,Z 708.225,A -85,B 0,C 180,E1 -7290,E2 -7290} C_VEL
LIN {X 0,Y 473.704,Z 707.979,A -85,B 0,C 180,E1 -7290.85,E2 -7290.85} C_VEL
LIN {X 0,Y 473.868,Z 706.282,A -85,B 0,C 180,E1 -7292.55,E2 -7292.55} C_VEL
LIN {X 0,Y 473.843,Z 704.803,A -85,B 0,C 180,E1 -7293.402,E2 -7293.402} C_VEL
LIN {X 0,Y 473.787,Z 701.717,A -85,B 0,C 180,E1 -7294.68,E2 -7294.68} C_VEL
LIN {X 0,Y 473.873,Z 697.559,A -85,B 0,C 180,E1 -7295.959,E2 -7295.959} C_VEL
LIN {X 0,Y 474.016,Z 691.162,A -85,B 0,C 180,E1 -7297.454,E2 -7297.454} C_VEL
LIN {X 0,Y 474.181,Z 684.186,A -85,B 0,C 180,E1 -7298.738,E2 -7298.738} C_VEL
LIN {X 0,Y 474.458,Z 675.522,A -85,B 0,C 180,E1 -7300.024,E2 -7300.024} C_VEL
LIN {X 0,Y 474.863,Z 665.598,A -85,B 0,C 180,E1 -7301.201,E2 -7301.201} C_VEL
LIN {X 0,Y 475.239,Z 656.258,A -85,B 0,C 180,E1 -7302.11,E2 -7302.11} C_VEL
LIN {X 0,Y 475.651,Z 644.726,A -85,B 0,C 180,E1 -7303.022,E2 -7303.022} C_VEL
LIN {X 0,Y 476.101,Z 632.516,A -85,B 0,C 180,E1 -7303.771,E2 -7303.771} C_VEL
LIN {X 0,Y 476.562,Z 619.855,A -85,B 0,C 180,E1 -7304.356,E2 -7304.356} C_VEL
LIN {X 0,Y 476.918,Z 607.713,A -85,B 0,C 180,E1 -7304.754,E2 -7304.754} C_VEL
LIN {X 0,Y 477.186,Z 592.859,A -85,B 0,C 180,E1 -7305.046,E2 -7305.046} C_VEL
LIN {X 0,Y 477.82,Z 513.177,A -85,B 0,C 180,E1 -7306.349,E2 -7306.349} C_VEL
LIN {X 0,Y 475.274,Z 492.779,A -85,B 0,C 180,E1 -7306.815,E2 -7306.815} C_VEL
LIN {X 0,Y 475.953,Z 471.256,A -85,B 0,C 180,E1 -7310.079,E2 -7310.079} C_VEL
LIN {X 0,Y 476.552,Z 455.262,A -85,B 0,C 180,E1 -7312.547,E2 -7312.547} C_VEL
LIN {X 0,Y 477.279,Z 437.897,A -85,B 0,C 180,E1 -7315.28,E2 -7315.28} C_VEL
LIN {X 0,Y 475.405,Z 427.723,A -85,B 0,C 180,E1 -7317.039,E2 -7317.039} C_VEL
LIN {X 0,Y 474.691,Z 424.359,A -85,B 0,C 180,E1 -7317.667,E2 -7317.667} C_VEL
LIN {X 0,Y 474.602,Z 424.373,A -85,B 0,C 180,E1 -7321.218,E2 -7321.218} C_VEL
LIN {X 0,Y 474.636,Z 424.365,A -85,B 0,C 180,E1 -7324.241,E2 -7324.241} C_VEL
LIN {X 0,Y 474.594,Z 424.368,A -85,B 0,C 180,E1 -7327.384,E2 -7327.384} C_VEL
LIN {X 0,Y 474.631,Z 424.361,A -85,B 0,C 180,E1 -7329.648,E2 -7329.648} C_VEL
LIN {X 0,Y 474.618,Z 424.367,A -85,B 0,C 180,E1 -7332.934,E2 -7332.934} C_VEL
LIN {X 0,Y 474.607,Z 424.362,A -85,B 0,C 180,E1 -7335.895,E2 -7335.895} C_VEL
LIN {X 0,Y 474.626,Z 424.363,A -85,B 0,C 180,E1 -7339.042,E2 -7339.042} C_VEL
LIN {X 0,Y 474.611,Z 424.362,A -85,B 0,C 180,E1 -7341.705,E2 -7341.705} C_VEL
LIN {X 0,Y 474.626,Z 424.364,A -85,B 0,C 180,E1 -7344.726,E2 -7344.726} C_VEL
LIN {X 0,Y 474.639,Z 424.358,A -85,B 0,C 180,E1 -7347.788,E2 -7347.788} C_VEL
LIN {X 0,Y 474.602,Z 424.365,A -85,B 0,C 180,E1 -7350.89,E2 -7350.89} C_VEL
LIN {X 0,Y 474.593,Z 424.365,A -85,B 0,C 180,E1 -7353.624,E2 -7353.624} C_VEL
LIN {X 0,Y 474.638,Z 424.362,A -85,B 0,C 180,E1 -7356.642,E2 -7356.642} C_VEL
LIN {X 0,Y 474.584,Z 424.371,A -85,B 0,C 180,E1 -7360.086,E2 -7360.086} C_VEL
LIN {X 0,Y 474.582,Z 424.367,A -85,B 0,C 180,E1 -7362.772,E2 -7362.772} C_VEL
LIN {X 0,Y 474.605,Z 424.365,A -85,B 0,C 180,E1 -7365.42,E2 -7365.42} C_VEL
LIN {X 0,Y 474.687,Z 424.359,A -85,B 0,C 180,E1 -7368.037,E2 -7368.037} C_VEL
LIN {X 0,Y 474.663,Z 424.361,A -85,B 0,C 180,E1 -7371.485,E2 -7371.485} C_VEL
LIN {X 0,Y 474.731,Z 424.354,A -85,B 0,C 180,E1 -7374.052,E2 -7374.052} C_VEL
LIN {X 0,Y 474.763,Z 424.532,A -85,B 0,C 180,E1 -7377.136,E2 -7377.136} C_VEL
LIN {X 0,Y 475.55,Z 428.975,A -85,B 0,C 180,E1 -7378.306,E2 -7378.306} C_VEL
LIN {X 0,Y 478.311,Z 439.556,A -85,B 0,C 180,E1 -7378.612,E2 -7378.612} C_VEL
LIN {X 0,Y 477.216,Z 534.934,A -85,B 0,C 180,E1 -7380.211,E2 -7380.211} C_VEL
LIN {X 0,Y 476.97,Z 548.92,A -85,B 0,C 180,E1 -7380.633,E2 -7380.633} C_VEL
LIN {X 0,Y 476.772,Z 560.751,A -85,B 0,C 180,E1 -7381.161,E2 -7381.161} C_VEL
LIN {X 0,Y 476.404,Z 573.102,A -85,B 0,C 180,E1 -7381.902,E2 -7381.902} C_VEL
LIN {X 0,Y 475.867,Z 584.212,A -85,B 0,C 180,E1 -7382.751,E2 -7382.751} C_VEL
LIN {X 0,Y 475.517,Z 593.182,A -85,B 0,C 180,E1 -7383.601,E2 -7383.601} C_VEL
LIN {X 0,Y 475.144,Z 602.403,A -85,B 0,C 180,E1 -7384.666,E2 -7384.666} C_VEL
LIN {X 0,Y 474.782,Z 611.33,A -85,B 0,C 180,E1 -7385.948,E2 -7385.948} C_VEL
LIN {X 0,Y 474.514,Z 618.677,A -85,B 0,C 180,E1 -7387.263,E2 -7387.263} C_VEL
LIN {X 0,Y 474.269,Z 624.265,A -85,B 0,C 180,E1 -7388.522,E2 -7388.522} C_VEL
LIN {X 0,Y 474.087,Z 628.764,A -85,B 0,C 180,E1 -7389.816,E2 -7389.816} C_VEL
LIN {X 0,Y 474.006,Z 632.155,A -85,B 0,C 180,E1 -7391.113,E2 -7391.113} C_VEL
LIN {X 0,Y 473.91,Z 633.834,A -85,B 0,C 180,E1 -7391.983,E2 -7391.983} C_VEL
LIN {X 0,Y 473.818,Z 635.101,A -85,B 0,C 180,E1 -7392.855,E2 -7392.855} C_VEL
LIN {X 0,Y 473.783,Z 635.94,A -85,B 0,C 180,E1 -7393.73,E2 -7393.73} C_VEL
LIN {X 0,Y 473.78,Z 636.308,A -85,B 0,C 180,E1 -7395.375,E2 -7395.375} C_VEL
LIN {X 0,Y 473.767,Z 635.839,A -85,B 0,C 180,E1 -7396.371,E2 -7396.371} C_VEL
LIN {X 0,Y 473.761,Z 634.918,A -85,B 0,C 180,E1 -7397.259,E2 -7397.259} C_VEL
LIN {X 0,Y 473.885,Z 633.203,A -85,B 0,C 180,E1 -7398.347,E2 -7398.347} C_VEL
LIN {X 0,Y 473.999,Z 629.399,A -85,B 0,C 180,E1 -7399.939,E2 -7399.939} C_VEL
LIN {X 0,Y 474.149,Z 624.858,A -85,B 0,C 180,E1 -7401.3,E2 -7401.3} C_VEL
LIN {X 0,Y 474.374,Z 618.993,A -85,B 0,C 180,E1 -7402.656,E2 -7402.656} C_VEL
LIN {X 0,Y 474.693,Z 611.471,A -85,B 0,C 180,E1 -7404.026,E2 -7404.026} C_VEL
LIN {X 0,Y 475.021,Z 603.626,A -85,B 0,C 180,E1 -7405.173,E2 -7405.173} C_VEL
LIN {X 0,Y 475.423,Z 593.955,A -85,B 0,C 180,E1 -7406.326,E2 -7406.326} C_VEL
LIN {X 0,Y 475.794,Z 584.411,A -85,B 0,C 180,E1 -7407.252,E2 -7407.252} C_VEL
LIN {X 0,Y 476.213,Z 573.606,A -85,B 0,C 180,E1 -7408.097,E2 -7408.097} C_VEL
LIN {X 0,Y 476.618,Z 561.915,A -85,B 0,C 180,E1 -7408.816,E2 -7408.816} C_VEL
LIN {X 0,Y 476.989,Z 549.035,A -85,B 0,C 180,E1 -7409.413,E2 -7409.413} C_VEL
LIN {X 0,Y 477.172,Z 536.568,A -85,B 0,C 180,E1 -7409.812,E2 -7409.812} C_VEL
LIN {X 0,Y 477.342,Z 519.535,A -85,B 0,C 180,E1 -7410.13,E2 -7410.13} C_VEL
LIN {X 0,Y 478.059,Z 439.01,A -85,B 0,C 180,E1 -7411.435,E2 -7411.435} C_VEL
LIN {X 0,Y 475.117,Z 426.793,A -85,B 0,C 180,E1 -7411.743,E2 -7411.743} C_VEL
LIN {X 0,Y 474.664,Z 424.362,A -85,B 0,C 180,E1 -7412.363,E2 -7412.363} C_VEL
LIN {X 0,Y 474.609,Z 424.362,A -85,B 0,C 180,E1 -7415.467,E2 -7415.467} C_VEL
LIN {X 0,Y 474.593,Z 424.37,A -85,B 0,C 180,E1 -7418.459,E2 -7418.459} C_VEL
LIN {X 0,Y 474.606,Z 424.362,A -85,B 0,C 180,E1 -7421.787,E2 -7421.787} C_VEL
LIN {X 0,Y 474.619,Z 424.364,A -85,B 0,C 180,E1 -7424.702,E2 -7424.702} C_VEL
LIN {X 0,Y 474.579,Z 424.365,A -85,B 0,C 180,E1 -7427.769,E2 -7427.769} C_VEL
